LIN {X 0,Y 516.535,Z 181.809,A -85,B 0,C 180,E1 -4926.761,E2 -4926.761} C_VEL
LIN {X 0,Y 516.469,Z 186.856,A -85,B 0,C 180,E1 -4929.874,E2 -4929.874} C_VEL
LIN {X 0,Y 516.401,Z 191.39,A -85,B 0,C 180,E1 -4932.578,E2 -4932.578} C_VEL
LIN {X 0,Y 516.332,Z 197.348,A -85,B 0,C 180,E1 -4936.019,E2 -4936.019} C_VEL
LIN {X 0,Y 516.35,Z 197.756,A -85,B 0,C 180,E1 -4936.183,E2 -4936.183} C_VEL
LIN {X 0,Y 518.498,Z 209.145,A -85,B 0,C 180,E1 -4936.528,E2 -4936.528} C_VEL
LIN {X 0,Y 518.233,Z 222.389,A -85,B 0,C 180,E1 -4937.02,E2 -4937.02} C_VEL
LIN {X 0,Y 517.941,Z 233.553,A -85,B 0,C 180,E1 -4937.583,E2 -4937.583} C_VEL
LIN {X 0,Y 517.678,Z 245.305,A -85,B 0,C 180,E1 -4938.35,E2 -4938.35} C_VEL
LIN {X 0,Y 517.363,Z 255.999,A -85,B 0,C 180,E1 -4939.235,E2 -4939.235} C_VEL
LIN {X 0,Y 517.09,Z 265.619,A -85,B 0,C 180,E1 -4940.219,E2 -4940.219} C_VEL
LIN {X 0,Y 516.888,Z 273.497,A -85,B 0,C 180,E1 -4941.202,E2 -4941.202} C_VEL
LIN {X 0,Y 516.632,Z 281.203,A -85,B 0,C 180,E1 -4942.378,E2 -4942.378} C_VEL
LIN {X 0,Y 516.521,Z 288.266,A -85,B 0,C 180,E1 -4943.751,E2 -4943.751} C_VEL
LIN {X 0,Y 516.313,Z 292.978,A -85,B 0,C 180,E1 -4944.924,E2 -4944.924} C_VEL
LIN {X 0,Y 516.373,Z 296.581,A -85,B 0,C 180,E1 -4946.098,E2 -4946.098} C_VEL
LIN {X 0,Y 516.327,Z 298.446,A -85,B 0,C 180,E1 -4946.879,E2 -4946.879} C_VEL
LIN {X 0,Y 516.266,Z 299.854,A -85,B 0,C 180,E1 -4947.66,E2 -4947.66} C_VEL
LIN {X 0,Y 516.162,Z 301.473,A -85,B 0,C 180,E1 -4949.22,E2 -4949.22} C_VEL
LIN {X 0,Y 516.158,Z 301.71,A -85,B 0,C 180,E1 -4950,E2 -4950} C_VEL
LIN {X 0,Y 516.162,Z 301.527,A -85,B 0,C 180,E1 -4950.78,E2 -4950.78} C_VEL
LIN {X 0,Y 516.266,Z 299.979,A -85,B 0,C 180,E1 -4952.341,E2 -4952.341} C_VEL
LIN {X 0,Y 516.327,Z 298.625,A -85,B 0,C 180,E1 -4953.121,E2 -4953.121} C_VEL
LIN {X 0,Y 516.366,Z 295.765,A -85,B 0,C 180,E1 -4954.293,E2 -4954.293} C_VEL
LIN {X 0,Y 516.406,Z 291.887,A -85,B 0,C 180,E1 -4955.467,E2 -4955.467} C_VEL
LIN {X 0,Y 516.501,Z 285.975,A -85,B 0,C 180,E1 -4956.826,E2 -4956.826} C_VEL
LIN {X 0,Y 516.689,Z 279.36,A -85,B 0,C 180,E1 -4958.014,E2 -4958.014} C_VEL
LIN {X 0,Y 516.918,Z 271.215,A -85,B 0,C 180,E1 -4959.193,E2 -4959.193} C_VEL
LIN {X 0,Y 517.183,Z 262.876,A -85,B 0,C 180,E1 -4960.175,E2 -4960.175} C_VEL
LIN {X 0,Y 517.449,Z 252.583,A -85,B 0,C 180,E1 -4961.16,E2 -4961.16} C_VEL
LIN {X 0,Y 517.786,Z 240.919,A -85,B 0,C 180,E1 -4962.049,E2 -4962.049} C_VEL
LIN {X 0,Y 518.096,Z 229.411,A -85,B 0,C 180,E1 -4962.735,E2 -4962.735} C_VEL
LIN {X 0,Y 518.366,Z 217.395,A -85,B 0,C 180,E1 -4963.276,E2 -4963.276} C_VEL
LIN {X 0,Y 518.295,Z 207.984,A -85,B 0,C 180,E1 -4963.602,E2 -4963.602} C_VEL
LIN {X 0,Y 516.35,Z 197.574,A -85,B 0,C 180,E1 -4963.931,E2 -4963.931} C_VEL
LIN {X 0,Y 516.402,Z 191.56,A -85,B 0,C 180,E1 -4967.422,E2 -4967.422} C_VEL
LIN {X 0,Y 516.456,Z 186.035,A -85,B 0,C 180,E1 -4970.721,E2 -4970.721} C_VEL
LIN {X 0,Y 516.533,Z 181.956,A -85,B 0,C 180,E1 -4973.24,E2 -4973.24} C_VEL
LIN {X 0,Y 516.595,Z 177.386,A -85,B 0,C 180,E1 -4976.117,E2 -4976.117} C_VEL
LIN {X 0,Y 516.706,Z 172.392,A -85,B 0,C 180,E1 -4979.318,E2 -4979.318} C_VEL
LIN {X 0,Y 516.761,Z 167.51,A -85,B 0,C 180,E1 -4982.519,E2 -4982.519} C_VEL
LIN {X 0,Y 516.796,Z 163.328,A -85,B 0,C 180,E1 -4985.318,E2 -4985.318} C_VEL
LIN {X 0,Y 516.855,Z 163.102,A -85,B 0,C 180,E1 -4987.939,E2 -4987.939} C_VEL
LIN {X 0,Y 516.855,Z 163.105,A -85,B 0,C 180,E1 -4990.744,E2 -4990.744} C_VEL
LIN {X 0,Y 516.859,Z 163.102,A -85,B 0,C 180,E1 -4992.834,E2 -4992.834} C_VEL
LIN {X 0,Y 516.897,Z 163.098,A -85,B 0,C 180,E1 -4995.007,E2 -4995.007} C_VEL
LIN {X 0,Y 516.915,Z 163.094,A -85,B 0,C 180,E1 -4998.399,E2 -4998.399} C_VEL
LIN {X 0,Y 516.877,Z 163.099,A -85,B 0,C 180,E1 -5001.283,E2 -5001.283} C_VEL
LIN {X 0,Y 516.852,Z 163.103,A -85,B 0,C 180,E1 -5004.673,E2 -5004.673} C_VEL
LIN {X 0,Y 516.895,Z 163.1,A -85,B 0,C 180,E1 -5007.457,E2 -5007.457} C_VEL
LIN {X 0,Y 516.923,Z 163.097,A -85,B 0,C 180,E1 -5010.695,E2 -5010.695} C_VEL
LIN {X 0,Y 516.944,Z 163.09,A -85,B 0,C 180,E1 -5013.804,E2 -5013.804} C_VEL
LIN {X 0,Y 516.859,Z 163.101,A -85,B 0,C 180,E1 -5016.776,E2 -5016.776} C_VEL
LIN {X 0,Y 516.94,Z 163.095,A -85,B 0,C 180,E1 -5019.732,E2 -5019.732} C_VEL
LIN {X 0,Y 516.908,Z 163.098,A -85,B 0,C 180,E1 -5022.595,E2 -5022.595} C_VEL
LIN {X 0,Y 516.944,Z 163.093,A -85,B 0,C 180,E1 -5025.03,E2 -5025.03} C_VEL
LIN {X 0,Y 516.967,Z 163.09,A -85,B 0,C 180,E1 -5028.234,E2 -5028.234} C_VEL
LIN {X 0,Y 516.93,Z 163.096,A -85,B 0,C 180,E1 -5031.399,E2 -5031.399} C_VEL
LIN {X 0,Y 517.008,Z 163.084,A -85,B 0,C 180,E1 -5034.54,E2 -5034.54} C_VEL
LIN {X 0,Y 517.08,Z 163.074,A -85,B 0,C 180,E1 -5037.663,E2 -5037.663} C_VEL
LIN {X 0,Y 517.095,Z 163.072,A -85,B 0,C 180,E1 -5040.779,E2 -5040.779} C_VEL
LIN {X 0,Y 517.011,Z 163.085,A -85,B 0,C 180,E1 -5043.117,E2 -5043.117} C_VEL
LIN {X 0,Y 516.973,Z 163.086,A -85,B 0,C 180,E1 -5046.244,E2 -5046.244} C_VEL
LIN {X 0,Y 516.933,Z 163.091,A -85,B 0,C 180,E1 -5049.39,E2 -5049.39} C_VEL
LIN {X 0,Y 516.985,Z 163.088,A -85,B 0,C 180,E1 -5051.824,E2 -5051.824} C_VEL
LIN {X 0,Y 516.946,Z 163.094,A -85,B 0,C 180,E1 -5055.146,E2 -5055.146} C_VEL
LIN {X 0,Y 516.917,Z 163.095,A -85,B 0,C 180,E1 -5058.223,E2 -5058.223} C_VEL
LIN {X 0,Y 516.913,Z 163.098,A -85,B 0,C 180,E1 -5060.702,E2 -5060.702} C_VEL
LIN {X 0,Y 516.89,Z 163.103,A -85,B 0,C 180,E1 -5064.073,E2 -5064.073} C_VEL
LIN {X 0,Y 516.923,Z 163.093,A -85,B 0,C 180,E1 -5066.658,E2 -5066.658} C_VEL
LIN {X 0,Y 516.912,Z 163.098,A -85,B 0,C 180,E1 -5069.524,E2 -5069.524} C_VEL
LIN {X 0,Y 516.897,Z 163.1,A -85,B 0,C 180,E1 -5072.543,E2 -5072.543} C_VEL
LIN {X 0,Y 516.854,Z 163.102,A -85,B 0,C 180,E1 -5075.328,E2 -5075.328} C_VEL
LIN {X 0,Y 516.872,Z 163.098,A -85,B 0,C 180,E1 -5078.717,E2 -5078.717} C_VEL
LIN {X 0,Y 516.913,Z 163.095,A -85,B 0,C 180,E1 -5081.775,E2 -5081.775} C_VEL
LIN {X 0,Y 516.896,Z 163.099,A -85,B 0,C 180,E1 -5085.007,E2 -5085.007} C_VEL
LIN {X 0,Y 516.915,Z 163.097,A -85,B 0,C 180,E1 -5088.399,E2 -5088.399} C_VEL
LIN {X 0,Y 516.877,Z 163.105,A -85,B 0,C 180,E1 -5091.284,E2 -5091.284} C_VEL
LIN {X 0,Y 516.893,Z 163.21,A -85,B 0,C 180,E1 -5092.277,E2 -5092.277} C_VEL
LIN {X 0,Y 517.603,Z 168.389,A -85,B 0,C 180,E1 -5094.556,E2 -5094.556} C_VEL
LIN {X 0,Y 517.467,Z 175.12,A -85,B 0,C 180,E1 -5097.358,E2 -5097.358} C_VEL
LIN {X 0,Y 517.281,Z 182.741,A -85,B 0,C 180,E1 -5100.405,E2 -5100.405} C_VEL
LIN {X 0,Y 517.087,Z 190.334,A -85,B 0,C 180,E1 -5103.351,E2 -5103.351} C_VEL
LIN {X 0,Y 516.934,Z 198.126,A -85,B 0,C 180,E1 -5106.355,E2 -5106.355} C_VEL
LIN {X 0,Y 516.785,Z 205.917,A -85,B 0,C 180,E1 -5109.293,E2 -5109.293} C_VEL
LIN {X 0,Y 516.635,Z 213.829,A -85,B 0,C 180,E1 -5112.221,E2 -5112.221} C_VEL
LIN {X 0,Y 516.548,Z 221.5,A -85,B 0,C 180,E1 -5115.018,E2 -5115.018} C_VEL
LIN {X 0,Y 516.504,Z 224.491,A -85,B 0,C 180,E1 -5116.099,E2 -5116.099} C_VEL
LIN {X 0,Y 518.468,Z 237.09,A -85,B 0,C 180,E1 -5116.452,E2 -5116.452} C_VEL
LIN {X 0,Y 518.229,Z 250.11,A -85,B 0,C 180,E1 -5116.92,E2 -5116.92} C_VEL
LIN {X 0,Y 517.912,Z 262.468,A -85,B 0,C 180,E1 -5117.533,E2 -5117.533} C_VEL
LIN {X 0,Y 517.621,Z 273.585,A -85,B 0,C 180,E1 -5118.249,E2 -5118.249} C_VEL
LIN {X 0,Y 517.322,Z 284.469,A -85,B 0,C 180,E1 -5119.135,E2 -5119.135} C_VEL
LIN {X 0,Y 517.038,Z 293.333,A -85,B 0,C 180,E1 -5120.02,E2 -5120.02} C_VEL
LIN {X 0,Y 516.814,Z 302.959,A -85,B 0,C 180,E1 -5121.2,E2 -5121.2} C_VEL
LIN {X 0,Y 516.563,Z 310.62,A -85,B 0,C 180,E1 -5122.377,E2 -5122.377} C_VEL
LIN {X 0,Y 516.427,Z 317.679,A -85,B 0,C 180,E1 -5123.75,E2 -5123.75} C_VEL
LIN {X 0,Y 516.313,Z 322.372,A -85,B 0,C 180,E1 -5124.924,E2 -5124.924} C_VEL
LIN {X 0,Y 516.355,Z 325.957,A -85,B 0,C 180,E1 -5126.098,E2 -5126.098} C_VEL
LIN {X 0,Y 516.282,Z 327.807,A -85,B 0,C 180,E1 -5126.878,E2 -5126.878} C_VEL
LIN {X 0,Y 516.261,Z 329.196,A -85,B 0,C 180,E1 -5127.659,E2 -5127.659} C_VEL
LIN {X 0,Y 516.16,Z 330.785,A -85,B 0,C 180,E1 -5129.22,E2 -5129.22} C_VEL
LIN {X 0,Y 516.154,Z 331,A -85,B 0,C 180,E1 -5130,E2 -5130} C_VEL
LIN {X 0,Y 516.192,Z 330.186,A -85,B 0,C 180,E1 -5131.56,E2 -5131.56} C_VEL
LIN {X 0,Y 516.261,Z 329.198,A -85,B 0,C 180,E1 -5132.34,E2 -5132.34} C_VEL
LIN {X 0,Y 516.282,Z 327.81,A -85,B 0,C 180,E1 -5133.121,E2 -5133.121} C_VEL
LIN {X 0,Y 516.343,Z 324.896,A -85,B 0,C 180,E1 -5134.293,E2 -5134.293} C_VEL
LIN {X 0,Y 516.405,Z 320.949,A -85,B 0,C 180,E1 -5135.466,E2 -5135.466} C_VEL
LIN {X 0,Y 516.487,Z 315.031,A -85,B 0,C 180,E1 -5136.808,E2 -5136.808} C_VEL
LIN {X 0,Y 516.64,Z 308.238,A -85,B 0,C 180,E1 -5138.015,E2 -5138.015} C_VEL
LIN {X 0,Y 516.867,Z 299.993,A -85,B 0,C 180,E1 -5139.193,E2 -5139.193} C_VEL
LIN {X 0,Y 517.076,Z 291.541,A -85,B 0,C 180,E1 -5140.177,E2 -5140.177} C_VEL
LIN {X 0,Y 517.44,Z 281.099,A -85,B 0,C 180,E1 -5141.16,E2 -5141.16} C_VEL
LIN {X 0,Y 517.705,Z 269.737,A -85,B 0,C 180,E1 -5142.019,E2 -5142.019} C_VEL
LIN {X 0,Y 517.977,Z 259.412,A -85,B 0,C 180,E1 -5142.638,E2 -5142.638} C_VEL
LIN {X 0,Y 518.279,Z 247.77,A -85,B 0,C 180,E1 -5143.178,E2 -5143.178} C_VEL
LIN {X 0,Y 518.366,Z 235.727,A -85,B 0,C 180,E1 -5143.588,E2 -5143.588} C_VEL
LIN {X 0,Y 516.504,Z 224.492,A -85,B 0,C 180,E1 -5143.901,E2 -5143.901} C_VEL
LIN {X 0,Y 516.615,Z 215.936,A -85,B 0,C 180,E1 -5147.006,E2 -5147.006} C_VEL
LIN {X 0,Y 516.791,Z 207.212,A -85,B 0,C 180,E1 -5150.223,E2 -5150.223} C_VEL
LIN {X 0,Y 516.909,Z 199.24,A -85,B 0,C 180,E1 -5153.221,E2 -5153.221} C_VEL
LIN {X 0,Y 517.077,Z 191.419,A -85,B 0,C 180,E1 -5156.226,E2 -5156.226} C_VEL
LIN {X 0,Y 517.262,Z 183.54,A -85,B 0,C 180,E1 -5159.283,E2 -5159.283} C_VEL
LIN {X 0,Y 517.402,Z 176.722,A -85,B 0,C 180,E1 -5161.988,E2 -5161.988} C_VEL
LIN {X 0,Y 517.61,Z 169.972,A -85,B 0,C 180,E1 -5164.768,E2 -5164.768} C_VEL
LIN {X 0,Y 517.286,Z 165.445,A -85,B 0,C 180,E1 -5166.717,E2 -5166.717} C_VEL
LIN {X 0,Y 516.878,Z 163.104,A -85,B 0,C 180,E1 -5167.8,E2 -5167.8} C_VEL
LIN {X 0,Y 516.882,Z 163.102,A -85,B 0,C 180,E1 -5170.741,E2 -5170.741} C_VEL
LIN {X 0,Y 516.883,Z 163.099,A -85,B 0,C 180,E1 -5172.831,E2 -5172.831} C_VEL
LIN {X 0,Y 516.894,Z 163.099,A -85,B 0,C 180,E1 -5175.007,E2 -5175.007} C_VEL
LIN {X 0,Y 516.912,Z 163.096,A -85,B 0,C 180,E1 -5178.398,E2 -5178.398} C_VEL
LIN {X 0,Y 516.873,Z 163.098,A -85,B 0,C 180,E1 -5181.283,E2 -5181.283} C_VEL
LIN {X 0,Y 516.853,Z 163.102,A -85,B 0,C 180,E1 -5184.672,E2 -5184.672} C_VEL
LIN {X 0,Y 516.894,Z 163.1,A -85,B 0,C 180,E1 -5187.456,E2 -5187.456} C_VEL
LIN {X 0,Y 516.921,Z 163.098,A -85,B 0,C 180,E1 -5190.695,E2 -5190.695} C_VEL
LIN {X 0,Y 516.941,Z 163.092,A -85,B 0,C 180,E1 -5193.804,E2 -5193.804} C_VEL
LIN {X 0,Y 516.856,Z 163.1,A -85,B 0,C 180,E1 -5196.776,E2 -5196.776} C_VEL
LIN {X 0,Y 516.937,Z 163.094,A -85,B 0,C 180,E1 -5199.732,E2 -5199.732} C_VEL
LIN {X 0,Y 516.919,Z 163.097,A -85,B 0,C 180,E1 -5202.596,E2 -5202.596} C_VEL
LIN {X 0,Y 516.94,Z 163.093,A -85,B 0,C 180,E1 -5205.03,E2 -5205.03} C_VEL
LIN {X 0,Y 516.964,Z 163.091,A -85,B 0,C 180,E1 -5208.234,E2 -5208.234} C_VEL
LIN {X 0,Y 516.926,Z 163.098,A -85,B 0,C 180,E1 -5211.399,E2 -5211.399} C_VEL
LIN {X 0,Y 517.01,Z 163.084,A -85,B 0,C 180,E1 -5214.54,E2 -5214.54} C_VEL
LIN {X 0,Y 517.08,Z 163.074,A -85,B 0,C 180,E1 -5217.663,E2 -5217.663} C_VEL
LIN {X 0,Y 517.092,Z 163.073,A -85,B 0,C 180,E1 -5220.779,E2 -5220.779} C_VEL
LIN {X 0,Y 517.008,Z 163.086,A -85,B 0,C 180,E1 -5223.117,E2 -5223.117} C_VEL
LIN {X 0,Y 516.969,Z 163.088,A -85,B 0,C 180,E1 -5226.244,E2 -5226.244} C_VEL
LIN {X 0,Y 516.934,Z 163.09,A -85,B 0,C 180,E1 -5229.39,E2 -5229.39} C_VEL
LIN {X 0,Y 516.95,Z 163.092,A -85,B 0,C 180,E1 -5231.807,E2 -5231.807} C_VEL
LIN {X 0,Y 516.943,Z 163.094,A -85,B 0,C 180,E1 -5235.147,E2 -5235.147} C_VEL
LIN {X 0,Y 516.923,Z 163.094,A -85,B 0,C 180,E1 -5238.222,E2 -5238.222} C_VEL
LIN {X 0,Y 516.91,Z 163.098,A -85,B 0,C 180,E1 -5240.702,E2 -5240.702} C_VEL
LIN {X 0,Y 516.888,Z 163.101,A -85,B 0,C 180,E1 -5244.073,E2 -5244.073} C_VEL
LIN {X 0,Y 516.924,Z 163.092,A -85,B 0,C 180,E1 -5246.658,E2 -5246.658} C_VEL
LIN {X 0,Y 516.91,Z 163.097,A -85,B 0,C 180,E1 -5249.524,E2 -5249.524} C_VEL
LIN {X 0,Y 516.894,Z 163.1,A -85,B 0,C 180,E1 -5252.544,E2 -5252.544} C_VEL
LIN {X 0,Y 516.853,Z 163.103,A -85,B 0,C 180,E1 -5255.328,E2 -5255.328} C_VEL
LIN {X 0,Y 516.874,Z 163.099,A -85,B 0,C 180,E1 -5258.717,E2 -5258.717} C_VEL
LIN {X 0,Y 516.911,Z 163.094,A -85,B 0,C 180,E1 -5261.776,E2 -5261.776} C_VEL
LIN {X 0,Y 516.923,Z 163.095,A -85,B 0,C 180,E1 -5265.01,E2 -5265.01} C_VEL
LIN {X 0,Y 516.913,Z 163.097,A -85,B 0,C 180,E1 -5268.399,E2 -5268.399} C_VEL
LIN {X 0,Y 516.861,Z 163.102,A -85,B 0,C 180,E1 -5270.288,E2 -5270.288} C_VEL
LIN {X 0,Y 516.201,Z 163.187,A -85,B 0,C 180,E1 -5270.939,E2 -5270.939} C_VEL
LIN {X 0,Y 513.362,Z 163.539,A -85,B 0,C 180,E1 -5271.994,E2 -5271.994} C_VEL
LIN {X 0,Y 510.94,Z 163.842,A -85,B 0,C 180,E1 -5272.845,E2 -5272.845} C_VEL
LIN {X 0,Y 509.871,Z 163.975,A -85,B 0,C 180,E1 -5273.501,E2 -5273.501} C_VEL
LIN {X 0,Y 509.769,Z 163.986,A -85,B 0,C 180,E1 -5273.724,E2 -5273.724} C_VEL
LIN {X 0,Y 509.728,Z 163.995,A -85,B 0,C 180,E1 -5274.614,E2 -5274.614} C_VEL
LIN {X 0,Y 509.723,Z 168.189,A -85,B 0,C 180,E1 -5277.471,E2 -5277.471} C_VEL
LIN {X 0,Y 509.636,Z 172.476,A -85,B 0,C 180,E1 -5280.318,E2 -5280.318} C_VEL
LIN {X 0,Y 509.553,Z 176.479,A -85,B 0,C 180,E1 -5282.926,E2 -5282.926} C_VEL
LIN {X 0,Y 509.555,Z 180.576,A -85,B 0,C 180,E1 -5285.558,E2 -5285.558} C_VEL
LIN {X 0,Y 509.424,Z 184.667,A -85,B 0,C 180,E1 -5288.131,E2 -5288.131} C_VEL
LIN {X 0,Y 509.328,Z 188.766,A -85,B 0,C 180,E1 -5290.661,E2 -5290.661} C_VEL
LIN {X 0,Y 509.278,Z 192.925,A -85,B 0,C 180,E1 -5293.154,E2 -5293.154} C_VEL
LIN {X 0,Y 509.251,Z 197.77,A -85,B 0,C 180,E1 -5295.974,E2 -5295.974} C_VEL
LIN {X 0,Y 511.595,Z 210.137,A -85,B 0,C 180,E1 -5296.368,E2 -5296.368} C_VEL
LIN {X 0,Y 511.296,Z 223.744,A -85,B 0,C 180,E1 -5296.892,E2 -5296.892} C_VEL
LIN {X 0,Y 511.018,Z 235.001,A -85,B 0,C 180,E1 -5297.482,E2 -5297.482} C_VEL
LIN {X 0,Y 510.737,Z 245.526,A -85,B 0,C 180,E1 -5298.189,E2 -5298.189} C_VEL
LIN {X 0,Y 510.398,Z 256.219,A -85,B 0,C 180,E1 -5299.086,E2 -5299.086} C_VEL
LIN {X 0,Y 510.098,Z 265.838,A -85,B 0,C 180,E1 -5300.083,E2 -5300.083} C_VEL
LIN {X 0,Y 509.88,Z 273.715,A -85,B 0,C 180,E1 -5301.08,E2 -5301.08} C_VEL
LIN {X 0,Y 509.603,Z 281.42,A -85,B 0,C 180,E1 -5302.273,E2 -5302.273} C_VEL
LIN {X 0,Y 509.443,Z 288.483,A -85,B 0,C 180,E1 -5303.664,E2 -5303.664} C_VEL
LIN {X 0,Y 509.248,Z 293.194,A -85,B 0,C 180,E1 -5304.854,E2 -5304.854} C_VEL
LIN {X 0,Y 509.305,Z 296.796,A -85,B 0,C 180,E1 -5306.044,E2 -5306.044} C_VEL
LIN {X 0,Y 509.241,Z 298.66,A -85,B 0,C 180,E1 -5306.836,E2 -5306.836} C_VEL
LIN {X 0,Y 509.196,Z 300.067,A -85,B 0,C 180,E1 -5307.627,E2 -5307.627} C_VEL
LIN {X 0,Y 509.076,Z 301.686,A -85,B 0,C 180,E1 -5309.209,E2 -5309.209} C_VEL
LIN {X 0,Y 509.069,Z 301.923,A -85,B 0,C 180,E1 -5310,E2 -5310} C_VEL
LIN {X 0,Y 509.075,Z 301.739,A -85,B 0,C 180,E1 -5310.791,E2 -5310.791} C_VEL
LIN {X 0,Y 509.196,Z 300.191,A -85,B 0,C 180,E1 -5312.373,E2 -5312.373} C_VEL
LIN {X 0,Y 509.242,Z 298.837,A -85,B 0,C 180,E1 -5313.165,E2 -5313.165} C_VEL
LIN {X 0,Y 509.289,Z 295.977,A -85,B 0,C 180,E1 -5314.353,E2 -5314.353} C_VEL
LIN {X 0,Y 509.351,Z 292.097,A -85,B 0,C 180,E1 -5315.543,E2 -5315.543} C_VEL
LIN {X 0,Y 509.431,Z 286.405,A -85,B 0,C 180,E1 -5316.878,E2 -5316.878} C_VEL
LIN {X 0,Y 509.655,Z 279.569,A -85,B 0,C 180,E1 -5318.126,E2 -5318.126} C_VEL
LIN {X 0,Y 509.911,Z 271.423,A -85,B 0,C 180,E1 -5319.32,E2 -5319.32} C_VEL
LIN {X 0,Y 510.181,Z 263.084,A -85,B 0,C 180,E1 -5320.316,E2 -5320.316} C_VEL
LIN {X 0,Y 510.491,Z 252.788,A -85,B 0,C 180,E1 -5321.314,E2 -5321.314} C_VEL
LIN {X 0,Y 510.819,Z 241.691,A -85,B 0,C 180,E1 -5322.175,E2 -5322.175} C_VEL
LIN {X 0,Y 511.135,Z 231.426,A -85,B 0,C 180,E1 -5322.81,E2 -5322.81} C_VEL
LIN {X 0,Y 511.41,Z 220.114,A -85,B 0,C 180,E1 -5323.359,E2 -5323.359} C_VEL
LIN {X 0,Y 511.429,Z 209.032,A -85,B 0,C 180,E1 -5323.763,E2 -5323.763} C_VEL
LIN {X 0,Y 509.273,Z 197.748,A -85,B 0,C 180,E1 -5324.128,E2 -5324.128} C_VEL
LIN {X 0,Y 509.352,Z 191.695,A -85,B 0,C 180,E1 -5327.671,E2 -5327.671} C_VEL
LIN {X 0,Y 509.399,Z 186.178,A -85,B 0,C 180,E1 -5331.021,E2 -5331.021} C_VEL
LIN {X 0,Y 509.471,Z 182.096,A -85,B 0,C 180,E1 -5333.581,E2 -5333.581} C_VEL
LIN {X 0,Y 509.53,Z 177.843,A -85,B 0,C 180,E1 -5336.291,E2 -5336.291} C_VEL
LIN {X 0,Y 509.61,Z 173.872,A -85,B 0,C 180,E1 -5338.861,E2 -5338.861} C_VEL
LIN {X 0,Y 509.661,Z 169.728,A -85,B 0,C 180,E1 -5341.601,E2 -5341.601} C_VEL
LIN {X 0,Y 509.759,Z 165.526,A -85,B 0,C 180,E1 -5344.421,E2 -5344.421} C_VEL
LIN {X 0,Y 509.761,Z 163.99,A -85,B 0,C 180,E1 -5345.568,E2 -5345.568} C_VEL
LIN {X 0,Y 509.811,Z 163.982,A -85,B 0,C 180,E1 -5348.342,E2 -5348.342} C_VEL
LIN {X 0,Y 509.837,Z 163.977,A -85,B 0,C 180,E1 -5351.427,E2 -5351.427} C_VEL
LIN {X 0,Y 509.841,Z 163.976,A -85,B 0,C 180,E1 -5354.67,E2 -5354.67} C_VEL
LIN {X 0,Y 509.857,Z 163.972,A -85,B 0,C 180,E1 -5358.103,E2 -5358.103} C_VEL
LIN {X 0,Y 509.846,Z 163.979,A -85,B 0,C 180,E1 -5360.647,E2 -5360.647} C_VEL
LIN {X 0,Y 509.78,Z 163.985,A -85,B 0,C 180,E1 -5363.643,E2 -5363.643} C_VEL
LIN {X 0,Y 509.84,Z 163.977,A -85,B 0,C 180,E1 -5366.537,E2 -5366.537} C_VEL
LIN {X 0,Y 509.847,Z 163.978,A -85,B 0,C 180,E1 -5369.334,E2 -5369.334} C_VEL
LIN {X 0,Y 509.894,Z 163.969,A -85,B 0,C 180,E1 -5372.054,E2 -5372.054} C_VEL
LIN {X 0,Y 509.841,Z 163.976,A -85,B 0,C 180,E1 -5374.702,E2 -5374.702} C_VEL
LIN {X 0,Y 509.826,Z 163.978,A -85,B 0,C 180,E1 -5377.458,E2 -5377.458} C_VEL
LIN {X 0,Y 509.918,Z 163.969,A -85,B 0,C 180,E1 -5379.845,E2 -5379.845} C_VEL
LIN {X 0,Y 509.876,Z 163.975,A -85,B 0,C 180,E1 -5383.174,E2 -5383.174} C_VEL
LIN {X 0,Y 509.865,Z 163.973,A -85,B 0,C 180,E1 -5385.634,E2 -5385.634} C_VEL
LIN {X 0,Y 509.912,Z 163.966,A -85,B 0,C 180,E1 -5388.874,E2 -5388.874} C_VEL
LIN {X 0,Y 509.876,Z 163.971,A -85,B 0,C 180,E1 -5392.077,E2 -5392.077} C_VEL
LIN {X 0,Y 509.959,Z 163.962,A -85,B 0,C 180,E1 -5394.464,E2 -5394.464} C_VEL
LIN {X 0,Y 510.052,Z 163.95,A -85,B 0,C 180,E1 -5397.631,E2 -5397.631} C_VEL
LIN {X 0,Y 510.065,Z 163.948,A -85,B 0,C 180,E1 -5400.789,E2 -5400.789} C_VEL
LIN {X 0,Y 509.952,Z 163.965,A -85,B 0,C 180,E1 -5403.16,E2 -5403.16} C_VEL
LIN {X 0,Y 509.921,Z 163.965,A -85,B 0,C 180,E1 -5406.33,E2 -5406.33} C_VEL
LIN {X 0,Y 509.874,Z 163.971,A -85,B 0,C 180,E1 -5409.521,E2 -5409.521} C_VEL
LIN {X 0,Y 509.953,Z 163.964,A -85,B 0,C 180,E1 -5411.931,E2 -5411.931} C_VEL
LIN {X 0,Y 509.895,Z 163.973,A -85,B 0,C 180,E1 -5415.242,E2 -5415.242} C_VEL
LIN {X 0,Y 509.868,Z 163.972,A -85,B 0,C 180,E1 -5417.993,E2 -5417.993} C_VEL
LIN {X 0,Y 509.887,Z 163.974,A -85,B 0,C 180,E1 -5420.401,E2 -5420.401} C_VEL
LIN {X 0,Y 509.822,Z 163.978,A -85,B 0,C 180,E1 -5423.564,E2 -5423.564} C_VEL
LIN {X 0,Y 509.91,Z 163.967,A -85,B 0,C 180,E1 -5426.378,E2 -5426.378} C_VEL
LIN {X 0,Y 509.877,Z 163.974,A -85,B 0,C 180,E1 -5428.844,E2 -5428.844} C_VEL
LIN {X 0,Y 509.821,Z 163.979,A -85,B 0,C 180,E1 -5431.59,E2 -5431.59} C_VEL
LIN {X 0,Y 509.846,Z 163.978,A -85,B 0,C 180,E1 -5434.414,E2 -5434.414} C_VEL
LIN {X 0,Y 509.78,Z 163.985,A -85,B 0,C 180,E1 -5437.344,E2 -5437.344} C_VEL
LIN {X 0,Y 509.838,Z 163.975,A -85,B 0,C 180,E1 -5440.382,E2 -5440.382} C_VEL
LIN {X 0,Y 509.824,Z 163.982,A -85,B 0,C 180,E1 -5443.062,E2 -5443.062} C_VEL
LIN {X 0,Y 509.824,Z 163.98,A -85,B 0,C 180,E1 -5445.793,E2 -5445.793} C_VEL
LIN {X 0,Y 509.857,Z 163.975,A -85,B 0,C 180,E1 -5448.575,E2 -5448.575} C_VEL
LIN {X 0,Y 509.853,Z 163.979,A -85,B 0,C 180,E1 -5451.975,E2 -5451.975} C_VEL
LIN {X 0,Y 510.431,Z 167.613,A -85,B 0,C 180,E1 -5453.697,E2 -5453.697} C_VEL
LIN {X 0,Y 510.577,Z 172.233,A -85,B 0,C 180,E1 -5455.679,E2 -5455.679} C_VEL
LIN {X 0,Y 510.368,Z 179.311,A -85,B 0,C 180,E1 -5458.624,E2 -5458.624} C_VEL
LIN {X 0,Y 510.186,Z 185.708,A -85,B 0,C 180,E1 -5461.175,E2 -5461.175} C_VEL
LIN {X 0,Y 510.005,Z 193.668,A -85,B 0,C 180,E1 -5464.273,E2 -5464.273} C_VEL
LIN {X 0,Y 509.847,Z 201.465,A -85,B 0,C 180,E1 -5467.296,E2 -5467.296} C_VEL
LIN {X 0,Y 509.712,Z 209.256,A -85,B 0,C 180,E1 -5470.256,E2 -5470.256} C_VEL
LIN {X 0,Y 509.507,Z 218.161,A -85,B 0,C 180,E1 -5473.574,E2 -5473.574} C_VEL
LIN {X 0,Y 509.443,Z 224.491,A -85,B 0,C 180,E1 -5475.902,E2 -5475.902} C_VEL
LIN {X 0,Y 511.562,Z 237.925,A -85,B 0,C 180,E1 -5476.291,E2 -5476.291} C_VEL
LIN {X 0,Y 511.291,Z 251.238,A -85,B 0,C 180,E1 -5476.79,E2 -5476.79} C_VEL
LIN {X 0,Y 510.959,Z 263.766,A -85,B 0,C 180,E1 -5477.436,E2 -5477.436} C_VEL
LIN {X 0,Y 510.62,Z 274.904,A -85,B 0,C 180,E1 -5478.186,E2 -5478.186} C_VEL
LIN {X 0,Y 510.295,Z 285.537,A -85,B 0,C 180,E1 -5479.084,E2 -5479.084} C_VEL
LIN {X 0,Y 510.002,Z 295.111,A -85,B 0,C 180,E1 -5480.081,E2 -5480.081} C_VEL
LIN {X 0,Y 509.76,Z 302.959,A -85,B 0,C 180,E1 -5481.077,E2 -5481.077} C_VEL
LIN {X 0,Y 509.522,Z 310.62,A -85,B 0,C 180,E1 -5482.271,E2 -5482.271} C_VEL
LIN {X 0,Y 509.336,Z 317.679,A -85,B 0,C 180,E1 -5483.662,E2 -5483.662} C_VEL
LIN {X 0,Y 509.248,Z 322.372,A -85,B 0,C 180,E1 -5484.853,E2 -5484.853} C_VEL
LIN {X 0,Y 509.253,Z 325.957,A -85,B 0,C 180,E1 -5486.043,E2 -5486.043} C_VEL
LIN {X 0,Y 509.2,Z 327.807,A -85,B 0,C 180,E1 -5486.835,E2 -5486.835} C_VEL
LIN {X 0,Y 509.161,Z 329.196,A -85,B 0,C 180,E1 -5487.627,E2 -5487.627} C_VEL
LIN {X 0,Y 509.073,Z 330.785,A -85,B 0,C 180,E1 -5489.209,E2 -5489.209} C_VEL
LIN {X 0,Y 509.065,Z 331,A -85,B 0,C 180,E1 -5490,E2 -5490} C_VEL
LIN {X 0,Y 509.112,Z 330.185,A -85,B 0,C 180,E1 -5491.582,E2 -5491.582} C_VEL
LIN {X 0,Y 509.161,Z 329.198,A -85,B 0,C 180,E1 -5492.373,E2 -5492.373} C_VEL
LIN {X 0,Y 509.2,Z 327.81,A -85,B 0,C 180,E1 -5493.165,E2 -5493.165} C_VEL
LIN {X 0,Y 509.234,Z 324.896,A -85,B 0,C 180,E1 -5494.353,E2 -5494.353} C_VEL
LIN {X 0,Y 509.345,Z 320.949,A -85,B 0,C 180,E1 -5495.542,E2 -5495.542} C_VEL
LIN {X 0,Y 509.41,Z 315.283,A -85,B 0,C 180,E1 -5496.853,E2 -5496.853} C_VEL
LIN {X 0,Y 509.585,Z 308.238,A -85,B 0,C 180,E1 -5498.127,E2 -5498.127} C_VEL
LIN {X 0,Y 509.846,Z 299.993,A -85,B 0,C 180,E1 -5499.321,E2 -5499.321} C_VEL
LIN {X 0,Y 510.065,Z 291.541,A -85,B 0,C 180,E1 -5500.318,E2 -5500.318} C_VEL
LIN {X 0,Y 510.468,Z 281.098,A -85,B 0,C 180,E1 -5501.314,E2 -5501.314} C_VEL
LIN {X 0,Y 510.737,Z 270.479,A -85,B 0,C 180,E1 -5502.133,E2 -5502.133} C_VEL
LIN {X 0,Y 511.049,Z 259.412,A -85,B 0,C 180,E1 -5502.812,E2 -5502.812} C_VEL
LIN {X 0,Y 511.371,Z 247.77,A -85,B 0,C 180,E1 -5503.359,E2 -5503.359} C_VEL
LIN {X 0,Y 511.408,Z 236.184,A -85,B 0,C 180,E1 -5503.763,E2 -5503.763} C_VEL
LIN {X 0,Y 509.442,Z 224.492,A -85,B 0,C 180,E1 -5504.097,E2 -5504.097} C_VEL
LIN {X 0,Y 509.541,Z 215.936,A -85,B 0,C 180,E1 -5507.25,E2 -5507.25} C_VEL
LIN {X 0,Y 509.731,Z 207.64,A -85,B 0,C 180,E1 -5510.353,E2 -5510.353} C_VEL
LIN {X 0,Y 509.888,Z 199.24,A -85,B 0,C 180,E1 -5513.56,E2 -5513.56} C_VEL
LIN {X 0,Y 510.037,Z 191.907,A -85,B 0,C 180,E1 -5516.406,E2 -5516.406} C_VEL
LIN {X 0,Y 510.24,Z 184.572,A -85,B 0,C 180,E1 -5519.273,E2 -5519.273} C_VEL
LIN {X 0,Y 510.392,Z 177.758,A -85,B 0,C 180,E1 -5522.014,E2 -5522.014} C_VEL
LIN {X 0,Y 510.618,Z 171.004,A -85,B 0,C 180,E1 -5524.833,E2 -5524.833} C_VEL
LIN {X 0,Y 510.454,Z 167.615,A -85,B 0,C 180,E1 -5526.301,E2 -5526.301} C_VEL
LIN {X 0,Y 509.851,Z 163.979,A -85,B 0,C 180,E1 -5528.024,E2 -5528.024} C_VEL
LIN {X 0,Y 509.855,Z 163.977,A -85,B 0,C 180,E1 -5531.425,E2 -5531.425} C_VEL
LIN {X 0,Y 509.838,Z 163.977,A -85,B 0,C 180,E1 -5534.67,E2 -5534.67} C_VEL
LIN {X 0,Y 509.854,Z 163.974,A -85,B 0,C 180,E1 -5538.103,E2 -5538.103} C_VEL
LIN {X 0,Y 509.842,Z 163.98,A -85,B 0,C 180,E1 -5540.647,E2 -5540.647} C_VEL
LIN {X 0,Y 509.778,Z 163.984,A -85,B 0,C 180,E1 -5543.643,E2 -5543.643} C_VEL
LIN {X 0,Y 509.856,Z 163.974,A -85,B 0,C 180,E1 -5546.539,E2 -5546.539} C_VEL
LIN {X 0,Y 509.844,Z 163.978,A -85,B 0,C 180,E1 -5549.334,E2 -5549.334} C_VEL
LIN {X 0,Y 509.892,Z 163.971,A -85,B 0,C 180,E1 -5552.054,E2 -5552.054} C_VEL
LIN {X 0,Y 509.838,Z 163.977,A -85,B 0,C 180,E1 -5554.702,E2 -5554.702} C_VEL
LIN {X 0,Y 509.823,Z 163.979,A -85,B 0,C 180,E1 -5557.458,E2 -5557.458} C_VEL
LIN {X 0,Y 509.914,Z 163.968,A -85,B 0,C 180,E1 -5559.845,E2 -5559.845} C_VEL
LIN {X 0,Y 509.88,Z 163.974,A -85,B 0,C 180,E1 -5563.175,E2 -5563.175} C_VEL
LIN {X 0,Y 509.862,Z 163.974,A -85,B 0,C 180,E1 -5565.634,E2 -5565.634} C_VEL
LIN {X 0,Y 509.909,Z 163.967,A -85,B 0,C 180,E1 -5568.874,E2 -5568.874} C_VEL
LIN {X 0,Y 509.873,Z 163.97,A -85,B 0,C 180,E1 -5572.077,E2 -5572.077} C_VEL
LIN {X 0,Y 509.96,Z 163.961,A -85,B 0,C 180,E1 -5574.464,E2 -5574.464} C_VEL
LIN {X 0,Y 510.051,Z 163.95,A -85,B 0,C 180,E1 -5577.631,E2 -5577.631} C_VEL
LIN {X 0,Y 510.062,Z 163.949,A -85,B 0,C 180,E1 -5580.79,E2 -5580.79} C_VEL
LIN {X 0,Y 509.95,Z 163.966,A -85,B 0,C 180,E1 -5583.16,E2 -5583.16} C_VEL
LIN {X 0,Y 509.917,Z 163.967,A -85,B 0,C 180,E1 -5586.33,E2 -5586.33} C_VEL
LIN {X 0,Y 509.875,Z 163.97,A -85,B 0,C 180,E1 -5589.521,E2 -5589.521} C_VEL
LIN {X 0,Y 509.902,Z 163.971,A -85,B 0,C 180,E1 -5591.932,E2 -5591.932} C_VEL
LIN {X 0,Y 509.892,Z 163.972,A -85,B 0,C 180,E1 -5595.242,E2 -5595.242} C_VEL
LIN {X 0,Y 509.88,Z 163.971,A -85,B 0,C 180,E1 -5597.999,E2 -5597.999} C_VEL
LIN {X 0,Y 509.848,Z 163.976,A -85,B 0,C 180,E1 -5601.002,E2 -5601.002} C_VEL
LIN {X 0,Y 509.819,Z 163.979,A -85,B 0,C 180,E1 -5603.564,E2 -5603.564} C_VEL
LIN {X 0,Y 509.91,Z 163.966,A -85,B 0,C 180,E1 -5606.379,E2 -5606.379} C_VEL
LIN {X 0,Y 509.875,Z 163.973,A -85,B 0,C 180,E1 -5608.845,E2 -5608.845} C_VEL
LIN {X 0,Y 509.819,Z 163.979,A -85,B 0,C 180,E1 -5611.59,E2 -5611.59} C_VEL
LIN {X 0,Y 509.843,Z 163.978,A -85,B 0,C 180,E1 -5614.414,E2 -5614.414} C_VEL
LIN {X 0,Y 509.781,Z 163.986,A -85,B 0,C 180,E1 -5617.344,E2 -5617.344} C_VEL
LIN {X 0,Y 509.837,Z 163.975,A -85,B 0,C 180,E1 -5620.383,E2 -5620.383} C_VEL
LIN {X 0,Y 509.822,Z 163.981,A -85,B 0,C 180,E1 -5623.062,E2 -5623.062} C_VEL
LIN {X 0,Y 509.83,Z 163.979,A -85,B 0,C 180,E1 -5625.793,E2 -5625.793} C_VEL
LIN {X 0,Y 509.855,Z 163.975,A -85,B 0,C 180,E1 -5628.575,E2 -5628.575} C_VEL
LIN {X 0,Y 509.847,Z 163.977,A -85,B 0,C 180,E1 -5631.787,E2 -5631.787} C_VEL
LIN {X 0,Y 509.769,Z 163.986,A -85,B 0,C 180,E1 -5633.724,E2 -5633.724} C_VEL
LIN {X 0,Y 509.056,Z 164.275,A -85,B 0,C 180,E1 -5634.382,E2 -5634.382} C_VEL
LIN {X 0,Y 506.184,Z 165.647,A -85,B 0,C 180,E1 -5635.441,E2 -5635.441} C_VEL
LIN {X 0,Y 503.773,Z 167.182,A -85,B 0,C 180,E1 -5636.291,E2 -5636.291} C_VEL
LIN {X 0,Y 502.732,Z 168.263,A -85,B 0,C 180,E1 -5636.948,E2 -5636.948} C_VEL
LIN {X 0,Y 502.642,Z 168.595,A -85,B 0,C 180,E1 -5637.171,E2 -5637.171} C_VEL
LIN {X 0,Y 502.588,Z 172.957,A -85,B 0,C 180,E1 -5640.111,E2 -5640.111} C_VEL
LIN {X 0,Y 502.519,Z 176.598,A -85,B 0,C 180,E1 -5642.515,E2 -5642.515} C_VEL
LIN {X 0,Y 502.49,Z 181.012,A -85,B 0,C 180,E1 -5645.384,E2 -5645.384} C_VEL
LIN {X 0,Y 502.389,Z 184.811,A -85,B 0,C 180,E1 -5647.809,E2 -5647.809} C_VEL
LIN {X 0,Y 502.29,Z 188.92,A -85,B 0,C 180,E1 -5650.379,E2 -5650.379} C_VEL
LIN {X 0,Y 502.223,Z 193.088,A -85,B 0,C 180,E1 -5652.911,E2 -5652.911} C_VEL
LIN {X 0,Y 502.195,Z 197.939,A -85,B 0,C 180,E1 -5655.772,E2 -5655.772} C_VEL
LIN {X 0,Y 504.719,Z 211.129,A -85,B 0,C 180,E1 -5656.205,E2 -5656.205} C_VEL
LIN {X 0,Y 504.384,Z 223.971,A -85,B 0,C 180,E1 -5656.709,E2 -5656.709} C_VEL
LIN {X 0,Y 504.084,Z 235.491,A -85,B 0,C 180,E1 -5657.324,E2 -5657.324} C_VEL
LIN {X 0,Y 503.759,Z 247.034,A -85,B 0,C 180,E1 -5658.125,E2 -5658.125} C_VEL
LIN {X 0,Y 503.395,Z 257.504,A -85,B 0,C 180,E1 -5659.035,E2 -5659.035} C_VEL
LIN {X 0,Y 503.111,Z 266.057,A -85,B 0,C 180,E1 -5659.944,E2 -5659.944} C_VEL
LIN {X 0,Y 502.868,Z 273.933,A -85,B 0,C 180,E1 -5660.954,E2 -5660.954} C_VEL
LIN {X 0,Y 502.549,Z 281.637,A -85,B 0,C 180,E1 -5662.163,E2 -5662.163} C_VEL
LIN {X 0,Y 502.361,Z 288.7,A -85,B 0,C 180,E1 -5663.574,E2 -5663.574} C_VEL
LIN {X 0,Y 502.187,Z 293.409,A -85,B 0,C 180,E1 -5664.781,E2 -5664.781} C_VEL
LIN {X 0,Y 502.238,Z 297.01,A -85,B 0,C 180,E1 -5665.988,E2 -5665.988} C_VEL
LIN {X 0,Y 502.16,Z 298.875,A -85,B 0,C 180,E1 -5666.791,E2 -5666.791} C_VEL
LIN {X 0,Y 502.128,Z 300.281,A -85,B 0,C 180,E1 -5667.594,E2 -5667.594} C_VEL
LIN {X 0,Y 501.992,Z 301.899,A -85,B 0,C 180,E1 -5669.198,E2 -5669.198} C_VEL
LIN {X 0,Y 501.984,Z 302.136,A -85,B 0,C 180,E1 -5670,E2 -5670} C_VEL
LIN {X 0,Y 501.992,Z 301.952,A -85,B 0,C 180,E1 -5670.802,E2 -5670.802} C_VEL
LIN {X 0,Y 502.128,Z 300.402,A -85,B 0,C 180,E1 -5672.407,E2 -5672.407} C_VEL
LIN {X 0,Y 502.16,Z 299.049,A -85,B 0,C 180,E1 -5673.209,E2 -5673.209} C_VEL
LIN {X 0,Y 502.214,Z 296.188,A -85,B 0,C 180,E1 -5674.414,E2 -5674.414} C_VEL
LIN {X 0,Y 502.299,Z 292.308,A -85,B 0,C 180,E1 -5675.621,E2 -5675.621} C_VEL
LIN {X 0,Y 502.356,Z 287.305,A -85,B 0,C 180,E1 -5676.829,E2 -5676.829} C_VEL
LIN {X 0,Y 502.58,Z 281.001,A -85,B 0,C 180,E1 -5678.039,E2 -5678.039} C_VEL
LIN {X 0,Y 502.827,Z 273.111,A -85,B 0,C 180,E1 -5679.25,E2 -5679.25} C_VEL
LIN {X 0,Y 503.163,Z 265.064,A -85,B 0,C 180,E1 -5680.259,E2 -5680.259} C_VEL
LIN {X 0,Y 503.468,Z 255.247,A -85,B 0,C 180,E1 -5681.27,E2 -5681.27} C_VEL
LIN {X 0,Y 503.8,Z 245.588,A -85,B 0,C 180,E1 -5682.079,E2 -5682.079} C_VEL
LIN {X 0,Y 504.08,Z 234.662,A -85,B 0,C 180,E1 -5682.816,E2 -5682.816} C_VEL
LIN {X 0,Y 504.457,Z 222.566,A -85,B 0,C 180,E1 -5683.444,E2 -5683.444} C_VEL
LIN {X 0,Y 504.608,Z 210.373,A -85,B 0,C 180,E1 -5683.914,E2 -5683.914} C_VEL
LIN {X 0,Y 502.202,Z 197.915,A -85,B 0,C 180,E1 -5684.331,E2 -5684.331} C_VEL
LIN {X 0,Y 502.255,Z 191.858,A -85,B 0,C 180,E1 -5687.929,E2 -5687.929} C_VEL
LIN {X 0,Y 502.325,Z 187.686,A -85,B 0,C 180,E1 -5690.474,E2 -5690.474} C_VEL
LIN {X 0,Y 502.393,Z 183.603,A -85,B 0,C 180,E1 -5693.06,E2 -5693.06} C_VEL
LIN {X 0,Y 502.445,Z 179.501,A -85,B 0,C 180,E1 -5695.697,E2 -5695.697} C_VEL
LIN {X 0,Y 502.558,Z 175.366,A -85,B 0,C 180,E1 -5698.39,E2 -5698.39} C_VEL
LIN {X 0,Y 502.606,Z 170.755,A -85,B 0,C 180,E1 -5701.463,E2 -5701.463} C_VEL
LIN {X 0,Y 502.714,Z 166.394,A -85,B 0,C 180,E1 -5704.429,E2 -5704.429} C_VEL
LIN {X 0,Y 502.736,Z 164.863,A -85,B 0,C 180,E1 -5705.824,E2 -5705.824} C_VEL
LIN {X 0,Y 502.778,Z 164.859,A -85,B 0,C 180,E1 -5708.978,E2 -5708.978} C_VEL
LIN {X 0,Y 502.776,Z 164.858,A -85,B 0,C 180,E1 -5712.195,E2 -5712.195} C_VEL
LIN {X 0,Y 502.788,Z 164.859,A -85,B 0,C 180,E1 -5715.47,E2 -5715.47} C_VEL
LIN {X 0,Y 502.821,Z 164.855,A -85,B 0,C 180,E1 -5718.934,E2 -5718.934} C_VEL
LIN {X 0,Y 502.762,Z 164.858,A -85,B 0,C 180,E1 -5722.043,E2 -5722.043} C_VEL
LIN {X 0,Y 502.787,Z 164.855,A -85,B 0,C 180,E1 -5725.033,E2 -5725.033} C_VEL
LIN {X 0,Y 502.784,Z 164.858,A -85,B 0,C 180,E1 -5727.915,E2 -5727.915} C_VEL
LIN {X 0,Y 502.826,Z 164.853,A -85,B 0,C 180,E1 -5730.712,E2 -5730.712} C_VEL
LIN {X 0,Y 502.864,Z 164.844,A -85,B 0,C 180,E1 -5733.439,E2 -5733.439} C_VEL
LIN {X 0,Y 502.776,Z 164.86,A -85,B 0,C 180,E1 -5736.085,E2 -5736.085} C_VEL
LIN {X 0,Y 502.784,Z 164.855,A -85,B 0,C 180,E1 -5738.689,E2 -5738.689} C_VEL
LIN {X 0,Y 502.827,Z 164.852,A -85,B 0,C 180,E1 -5741.248,E2 -5741.248} C_VEL
LIN {X 0,Y 502.85,Z 164.849,A -85,B 0,C 180,E1 -5744.6,E2 -5744.6} C_VEL
LIN {X 0,Y 502.878,Z 164.847,A -85,B 0,C 180,E1 -5748.039,E2 -5748.039} C_VEL
LIN {X 0,Y 502.85,Z 164.847,A -85,B 0,C 180,E1 -5751.156,E2 -5751.156} C_VEL
LIN {X 0,Y 502.912,Z 164.839,A -85,B 0,C 180,E1 -5754.386,E2 -5754.386} C_VEL
LIN {X 0,Y 503.022,Z 164.826,A -85,B 0,C 180,E1 -5757.598,E2 -5757.598} C_VEL
LIN {X 0,Y 503.029,Z 164.827,A -85,B 0,C 180,E1 -5760,E2 -5760} C_VEL
LIN {X 0,Y 503.024,Z 164.825,A -85,B 0,C 180,E1 -5762.402,E2 -5762.402} C_VEL
LIN {X 0,Y 502.916,Z 164.838,A -85,B 0,C 180,E1 -5765.614,E2 -5765.614} C_VEL
LIN {X 0,Y 502.847,Z 164.85,A -85,B 0,C 180,E1 -5768.844,E2 -5768.844} C_VEL
LIN {X 0,Y 502.895,Z 164.844,A -85,B 0,C 180,E1 -5772.1,E2 -5772.1} C_VEL
LIN {X 0,Y 502.85,Z 164.849,A -85,B 0,C 180,E1 -5775.4,E2 -5775.4} C_VEL
LIN {X 0,Y 502.827,Z 164.854,A -85,B 0,C 180,E1 -5778.752,E2 -5778.752} C_VEL
LIN {X 0,Y 502.784,Z 164.854,A -85,B 0,C 180,E1 -5781.311,E2 -5781.311} C_VEL
LIN {X 0,Y 502.775,Z 164.859,A -85,B 0,C 180,E1 -5783.915,E2 -5783.915} C_VEL
LIN {X 0,Y 502.865,Z 164.844,A -85,B 0,C 180,E1 -5786.566,E2 -5786.566} C_VEL
LIN {X 0,Y 502.825,Z 164.853,A -85,B 0,C 180,E1 -5789.288,E2 -5789.288} C_VEL
LIN {X 0,Y 502.784,Z 164.857,A -85,B 0,C 180,E1 -5792.085,E2 -5792.085} C_VEL
LIN {X 0,Y 502.791,Z 164.854,A -85,B 0,C 180,E1 -5794.967,E2 -5794.967} C_VEL
LIN {X 0,Y 502.763,Z 164.856,A -85,B 0,C 180,E1 -5798.481,E2 -5798.481} C_VEL
LIN {X 0,Y 502.821,Z 164.853,A -85,B 0,C 180,E1 -5801.066,E2 -5801.066} C_VEL
LIN {X 0,Y 502.787,Z 164.859,A -85,B 0,C 180,E1 -5804.53,E2 -5804.53} C_VEL
LIN {X 0,Y 502.796,Z 164.855,A -85,B 0,C 180,E1 -5807.861,E2 -5807.861} C_VEL
LIN {X 0,Y 502.78,Z 164.859,A -85,B 0,C 180,E1 -5810.247,E2 -5810.247} C_VEL
LIN {X 0,Y 502.841,Z 164.998,A -85,B 0,C 180,E1 -5811.918,E2 -5811.918} C_VEL
LIN {X 0,Y 503.524,Z 169.766,A -85,B 0,C 180,E1 -5814.111,E2 -5814.111} C_VEL
LIN {X 0,Y 503.547,Z 174.308,A -85,B 0,C 180,E1 -5816.063,E2 -5816.063} C_VEL
LIN {X 0,Y 503.311,Z 181.041,A -85,B 0,C 180,E1 -5818.892,E2 -5818.892} C_VEL
LIN {X 0,Y 503.147,Z 187.878,A -85,B 0,C 180,E1 -5821.646,E2 -5821.646} C_VEL
LIN {X 0,Y 502.967,Z 195.814,A -85,B 0,C 180,E1 -5824.775,E2 -5824.775} C_VEL
LIN {X 0,Y 502.768,Z 203.691,A -85,B 0,C 180,E1 -5827.826,E2 -5827.826} C_VEL
LIN {X 0,Y 502.593,Z 211.482,A -85,B 0,C 180,E1 -5830.815,E2 -5830.815} C_VEL
LIN {X 0,Y 502.441,Z 219.274,A -85,B 0,C 180,E1 -5833.754,E2 -5833.754} C_VEL
LIN {X 0,Y 502.367,Z 224.491,A -85,B 0,C 180,E1 -5835.699,E2 -5835.699} C_VEL
LIN {X 0,Y 504.625,Z 237.925,A -85,B 0,C 180,E1 -5836.099,E2 -5836.099} C_VEL
LIN {X 0,Y 504.398,Z 251.238,A -85,B 0,C 180,E1 -5836.606,E2 -5836.606} C_VEL
LIN {X 0,Y 504.029,Z 262.609,A -85,B 0,C 180,E1 -5837.192,E2 -5837.192} C_VEL
LIN {X 0,Y 503.711,Z 273.586,A -85,B 0,C 180,E1 -5837.919,E2 -5837.919} C_VEL
LIN {X 0,Y 503.371,Z 284.467,A -85,B 0,C 180,E1 -5838.83,E2 -5838.83} C_VEL
LIN {X 0,Y 503.023,Z 293.332,A -85,B 0,C 180,E1 -5839.739,E2 -5839.739} C_VEL
LIN {X 0,Y 502.704,Z 302.959,A -85,B 0,C 180,E1 -5840.951,E2 -5840.951} C_VEL
LIN {X 0,Y 502.47,Z 310.621,A -85,B 0,C 180,E1 -5842.162,E2 -5842.162} C_VEL
LIN {X 0,Y 502.275,Z 317.679,A -85,B 0,C 180,E1 -5843.573,E2 -5843.573} C_VEL
LIN {X 0,Y 502.186,Z 322.372,A -85,B 0,C 180,E1 -5844.781,E2 -5844.781} C_VEL
LIN {X 0,Y 502.152,Z 325.958,A -85,B 0,C 180,E1 -5845.987,E2 -5845.987} C_VEL
LIN {X 0,Y 502.121,Z 327.807,A -85,B 0,C 180,E1 -5846.79,E2 -5846.79} C_VEL
LIN {X 0,Y 502.066,Z 329.195,A -85,B 0,C 180,E1 -5847.593,E2 -5847.593} C_VEL
LIN {X 0,Y 501.99,Z 330.786,A -85,B 0,C 180,E1 -5849.198,E2 -5849.198} C_VEL
LIN {X 0,Y 501.98,Z 331,A -85,B 0,C 180,E1 -5850,E2 -5850} C_VEL
LIN {X 0,Y 502.036,Z 330.185,A -85,B 0,C 180,E1 -5851.604,E2 -5851.604} C_VEL
LIN {X 0,Y 502.066,Z 329.198,A -85,B 0,C 180,E1 -5852.407,E2 -5852.407} C_VEL
LIN {X 0,Y 502.121,Z 327.81,A -85,B 0,C 180,E1 -5853.209,E2 -5853.209} C_VEL
LIN {X 0,Y 502.128,Z 324.896,A -85,B 0,C 180,E1 -5854.415,E2 -5854.415} C_VEL
LIN {X 0,Y 502.26,Z 320.949,A -85,B 0,C 180,E1 -5855.621,E2 -5855.621} C_VEL
LIN {X 0,Y 502.335,Z 314.978,A -85,B 0,C 180,E1 -5857.011,E2 -5857.011} C_VEL
LIN {X 0,Y 502.542,Z 308.238,A -85,B 0,C 180,E1 -5858.241,E2 -5858.241} C_VEL
LIN {X 0,Y 502.811,Z 299.993,A -85,B 0,C 180,E1 -5859.453,E2 -5859.453} C_VEL
LIN {X 0,Y 503.058,Z 291.541,A -85,B 0,C 180,E1 -5860.464,E2 -5860.464} C_VEL
LIN {X 0,Y 503.495,Z 281.097,A -85,B 0,C 180,E1 -5861.473,E2 -5861.473} C_VEL
LIN {X 0,Y 503.794,Z 269.422,A -85,B 0,C 180,E1 -5862.378,E2 -5862.378} C_VEL
LIN {X 0,Y 504.159,Z 257.494,A -85,B 0,C 180,E1 -5863.092,E2 -5863.092} C_VEL
LIN {X 0,Y 504.545,Z 245.173,A -85,B 0,C 180,E1 -5863.646,E2 -5863.646} C_VEL
LIN {X 0,Y 504.416,Z 236.64,A -85,B 0,C 180,E1 -5863.945,E2 -5863.945} C_VEL
LIN {X 0,Y 502.366,Z 224.492,A -85,B 0,C 180,E1 -5864.3,E2 -5864.3} C_VEL
LIN {X 0,Y 502.467,Z 217.049,A -85,B 0,C 180,E1 -5867.081,E2 -5867.081} C_VEL
LIN {X 0,Y 502.661,Z 209.257,A -85,B 0,C 180,E1 -5870.032,E2 -5870.032} C_VEL
LIN {X 0,Y 502.837,Z 201.466,A -85,B 0,C 180,E1 -5873.038,E2 -5873.038} C_VEL
LIN {X 0,Y 502.975,Z 193.541,A -85,B 0,C 180,E1 -5876.113,E2 -5876.113} C_VEL
LIN {X 0,Y 503.157,Z 186.742,A -85,B 0,C 180,E1 -5878.808,E2 -5878.808} C_VEL
LIN {X 0,Y 503.406,Z 179.817,A -85,B 0,C 180,E1 -5881.612,E2 -5881.612} C_VEL
LIN {X 0,Y 503.628,Z 172.034,A -85,B 0,C 180,E1 -5884.9,E2 -5884.9} C_VEL
LIN {X 0,Y 503.271,Z 167.521,A -85,B 0,C 180,E1 -5886.904,E2 -5886.904} C_VEL
LIN {X 0,Y 502.816,Z 164.856,A -85,B 0,C 180,E1 -5888.217,E2 -5888.217} C_VEL
LIN {X 0,Y 502.819,Z 164.853,A -85,B 0,C 180,E1 -5891.066,E2 -5891.066} C_VEL
LIN {X 0,Y 502.785,Z 164.855,A -85,B 0,C 180,E1 -5894.53,E2 -5894.53} C_VEL
LIN {X 0,Y 502.794,Z 164.853,A -85,B 0,C 180,E1 -5897.86,E2 -5897.86} C_VEL
LIN {X 0,Y 502.786,Z 164.856,A -85,B 0,C 180,E1 -5900.245,E2 -5900.245} C_VEL
LIN {X 0,Y 502.718,Z 164.862,A -85,B 0,C 180,E1 -5903.048,E2 -5903.048} C_VEL
LIN {X 0,Y 502.801,Z 164.856,A -85,B 0,C 180,E1 -5906.006,E2 -5906.006} C_VEL
LIN {X 0,Y 502.794,Z 164.857,A -85,B 0,C 180,E1 -5908.857,E2 -5908.857} C_VEL
LIN {X 0,Y 502.843,Z 164.848,A -85,B 0,C 180,E1 -5911.705,E2 -5911.705} C_VEL
LIN {X 0,Y 502.82,Z 164.854,A -85,B 0,C 180,E1 -5914.323,E2 -5914.323} C_VEL
LIN {X 0,Y 502.8,Z 164.853,A -85,B 0,C 180,E1 -5917.298,E2 -5917.298} C_VEL
LIN {X 0,Y 502.822,Z 164.85,A -85,B 0,C 180,E1 -5920.4,E2 -5920.4} C_VEL
LIN {X 0,Y 502.828,Z 164.852,A -85,B 0,C 180,E1 -5922.931,E2 -5922.931} C_VEL
LIN {X 0,Y 502.843,Z 164.848,A -85,B 0,C 180,E1 -5925.429,E2 -5925.429} C_VEL
LIN {X 0,Y 502.873,Z 164.844,A -85,B 0,C 180,E1 -5928.717,E2 -5928.717} C_VEL
LIN {X 0,Y 502.845,Z 164.846,A -85,B 0,C 180,E1 -5931.966,E2 -5931.966} C_VEL
LIN {X 0,Y 502.913,Z 164.838,A -85,B 0,C 180,E1 -5934.386,E2 -5934.386} C_VEL
LIN {X 0,Y 503.021,Z 164.826,A -85,B 0,C 180,E1 -5937.598,E2 -5937.598} C_VEL
LIN {X 0,Y 503.026,Z 164.827,A -85,B 0,C 180,E1 -5940,E2 -5940} C_VEL
LIN {X 0,Y 503.02,Z 164.826,A -85,B 0,C 180,E1 -5942.402,E2 -5942.402} C_VEL
LIN {X 0,Y 502.912,Z 164.84,A -85,B 0,C 180,E1 -5945.614,E2 -5945.614} C_VEL
LIN {X 0,Y 502.846,Z 164.848,A -85,B 0,C 180,E1 -5948.844,E2 -5948.844} C_VEL
LIN {X 0,Y 502.844,Z 164.852,A -85,B 0,C 180,E1 -5952.102,E2 -5952.102} C_VEL
LIN {X 0,Y 502.847,Z 164.85,A -85,B 0,C 180,E1 -5955.4,E2 -5955.4} C_VEL
LIN {X 0,Y 502.839,Z 164.849,A -85,B 0,C 180,E1 -5958.12,E2 -5958.12} C_VEL
LIN {X 0,Y 502.827,Z 164.853,A -85,B 0,C 180,E1 -5960.536,E2 -5960.536} C_VEL
LIN {X 0,Y 502.785,Z 164.854,A -85,B 0,C 180,E1 -5963.041,E2 -5963.041} C_VEL
LIN {X 0,Y 502.82,Z 164.855,A -85,B 0,C 180,E1 -5965.677,E2 -5965.677} C_VEL
LIN {X 0,Y 502.839,Z 164.848,A -85,B 0,C 180,E1 -5968.373,E2 -5968.373} C_VEL
LIN {X 0,Y 502.791,Z 164.855,A -85,B 0,C 180,E1 -5971.499,E2 -5971.499} C_VEL
LIN {X 0,Y 502.801,Z 164.857,A -85,B 0,C 180,E1 -5973.994,E2 -5973.994} C_VEL
LIN {X 0,Y 502.735,Z 164.862,A -85,B 0,C 180,E1 -5977.172,E2 -5977.172} C_VEL
LIN {X 0,Y 502.786,Z 164.853,A -85,B 0,C 180,E1 -5980.016,E2 -5980.016} C_VEL
LIN {X 0,Y 502.802,Z 164.852,A -85,B 0,C 180,E1 -5982.2,E2 -5982.2} C_VEL
LIN {X 0,Y 502.801,Z 164.853,A -85,B 0,C 180,E1 -5985.469,E2 -5985.469} C_VEL
LIN {X 0,Y 502.819,Z 164.851,A -85,B 0,C 180,E1 -5988.934,E2 -5988.934} C_VEL
LIN {X 0,Y 502.787,Z 164.855,A -85,B 0,C 180,E1 -5992.046,E2 -5992.046} C_VEL
LIN {X 0,Y 502.696,Z 164.867,A -85,B 0,C 180,E1 -5994.182,E2 -5994.182} C_VEL
LIN {X 0,Y 502.665,Z 165.48,A -85,B 0,C 180,E1 -5995.024,E2 -5995.024} C_VEL
LIN {X 0,Y 502.642,Z 168.595,A -85,B 0,C 180,E1 -5997.171,E2 -5997.171} C_VEL
LIN {X 0,Y 501.959,Z 169.639,A -85,B 0,C 180,E1 -5997.829,E2 -5997.829} C_VEL
LIN {X 0,Y 499.084,Z 171.549,A -85,B 0,C 180,E1 -5998.893,E2 -5998.893} C_VEL
LIN {X 0,Y 496.653,Z 173.1,A -85,B 0,C 180,E1 -5999.75,E2 -5999.75} C_VEL
LIN {X 0,Y 495.598,Z 174.206,A -85,B 0,C 180,E1 -6000.413,E2 -6000.413} C_VEL
LIN {X 0,Y 495.507,Z 174.55,A -85,B 0,C 180,E1 -6000.639,E2 -6000.639} C_VEL
LIN {X 0,Y 495.438,Z 178.613,A -85,B 0,C 180,E1 -6003.34,E2 -6003.34} C_VEL
LIN {X 0,Y 495.394,Z 182.222,A -85,B 0,C 180,E1 -6005.707,E2 -6005.707} C_VEL
LIN {X 0,Y 495.291,Z 186.328,A -85,B 0,C 180,E1 -6008.351,E2 -6008.351} C_VEL
LIN {X 0,Y 495.196,Z 190.468,A -85,B 0,C 180,E1 -6010.948,E2 -6010.948} C_VEL
LIN {X 0,Y 495.118,Z 194.661,A -85,B 0,C 180,E1 -6013.508,E2 -6013.508} C_VEL
LIN {X 0,Y 495.13,Z 198.133,A -85,B 0,C 180,E1 -6015.565,E2 -6015.565} C_VEL
LIN {X 0,Y 497.831,Z 212.119,A -85,B 0,C 180,E1 -6016.036,E2 -6016.036} C_VEL
LIN {X 0,Y 497.472,Z 225.307,A -85,B 0,C 180,E1 -6016.572,E2 -6016.572} C_VEL
LIN {X 0,Y 497.157,Z 237.166,A -85,B 0,C 180,E1 -6017.239,E2 -6017.239} C_VEL
LIN {X 0,Y 496.788,Z 248.54,A -85,B 0,C 180,E1 -6018.06,E2 -6018.06} C_VEL
LIN {X 0,Y 496.392,Z 258.784,A -85,B 0,C 180,E1 -6018.981,E2 -6018.981} C_VEL
LIN {X 0,Y 496.036,Z 267.974,A -85,B 0,C 180,E1 -6020.005,E2 -6020.005} C_VEL
LIN {X 0,Y 495.723,Z 276.892,A -85,B 0,C 180,E1 -6021.234,E2 -6021.234} C_VEL
LIN {X 0,Y 495.431,Z 284.073,A -85,B 0,C 180,E1 -6022.46,E2 -6022.46} C_VEL
LIN {X 0,Y 495.292,Z 288.916,A -85,B 0,C 180,E1 -6023.482,E2 -6023.482} C_VEL
LIN {X 0,Y 495.13,Z 293.624,A -85,B 0,C 180,E1 -6024.706,E2 -6024.706} C_VEL
LIN {X 0,Y 495.153,Z 297.225,A -85,B 0,C 180,E1 -6025.931,E2 -6025.931} C_VEL
LIN {X 0,Y 495.083,Z 299.089,A -85,B 0,C 180,E1 -6026.745,E2 -6026.745} C_VEL
LIN {X 0,Y 495.033,Z 300.495,A -85,B 0,C 180,E1 -6027.559,E2 -6027.559} C_VEL
LIN {X 0,Y 494.912,Z 302.112,A -85,B 0,C 180,E1 -6029.187,E2 -6029.187} C_VEL
LIN {X 0,Y 494.901,Z 302.348,A -85,B 0,C 180,E1 -6030,E2 -6030} C_VEL
LIN {X 0,Y 494.912,Z 302.164,A -85,B 0,C 180,E1 -6030.814,E2 -6030.814} C_VEL
LIN {X 0,Y 495.033,Z 300.614,A -85,B 0,C 180,E1 -6032.441,E2 -6032.441} C_VEL
LIN {X 0,Y 495.083,Z 299.26,A -85,B 0,C 180,E1 -6033.255,E2 -6033.255} C_VEL
LIN {X 0,Y 495.122,Z 296.4,A -85,B 0,C 180,E1 -6034.478,E2 -6034.478} C_VEL
LIN {X 0,Y 495.248,Z 292.518,A -85,B 0,C 180,E1 -6035.701,E2 -6035.701} C_VEL
LIN {X 0,Y 495.309,Z 287.515,A -85,B 0,C 180,E1 -6036.927,E2 -6036.927} C_VEL
LIN {X 0,Y 495.536,Z 281.211,A -85,B 0,C 180,E1 -6038.154,E2 -6038.154} C_VEL
LIN {X 0,Y 495.817,Z 273.319,A -85,B 0,C 180,E1 -6039.382,E2 -6039.382} C_VEL
LIN {X 0,Y 496.172,Z 265.272,A -85,B 0,C 180,E1 -6040.405,E2 -6040.405} C_VEL
LIN {X 0,Y 496.501,Z 255.453,A -85,B 0,C 180,E1 -6041.43,E2 -6041.43} C_VEL
LIN {X 0,Y 496.887,Z 244.551,A -85,B 0,C 180,E1 -6042.343,E2 -6042.343} C_VEL
LIN {X 0,Y 497.226,Z 233.592,A -85,B 0,C 180,E1 -6043.071,E2 -6043.071} C_VEL
LIN {X 0,Y 497.6,Z 221.639,A -85,B 0,C 180,E1 -6043.685,E2 -6043.685} C_VEL
LIN {X 0,Y 497.657,Z 210.951,A -85,B 0,C 180,E1 -6044.1,E2 -6044.1} C_VEL
LIN {X 0,Y 495.114,Z 198.108,A -85,B 0,C 180,E1 -6044.541,E2 -6044.541} C_VEL
LIN {X 0,Y 495.193,Z 192.293,A -85,B 0,C 180,E1 -6048.029,E2 -6048.029} C_VEL
LIN {X 0,Y 495.242,Z 187.842,A -85,B 0,C 180,E1 -6050.78,E2 -6050.78} C_VEL
LIN {X 0,Y 495.321,Z 183.742,A -85,B 0,C 180,E1 -6053.409,E2 -6053.409} C_VEL
LIN {X 0,Y 495.396,Z 181.002,A -85,B 0,C 180,E1 -6055.189,E2 -6055.189} C_VEL
LIN {X 0,Y 495.511,Z 176.079,A -85,B 0,C 180,E1 -6058.433,E2 -6058.433} C_VEL
LIN {X 0,Y 495.565,Z 171.308,A -85,B 0,C 180,E1 -6061.65,E2 -6061.65} C_VEL
LIN {X 0,Y 495.686,Z 166.92,A -85,B 0,C 180,E1 -6064.679,E2 -6064.679} C_VEL
LIN {X 0,Y 495.641,Z 165.749,A -85,B 0,C 180,E1 -6065.547,E2 -6065.547} C_VEL
LIN {X 0,Y 495.736,Z 165.736,A -85,B 0,C 180,E1 -6068.764,E2 -6068.764} C_VEL
LIN {X 0,Y 495.745,Z 165.735,A -85,B 0,C 180,E1 -6071.782,E2 -6071.782} C_VEL
LIN {X 0,Y 495.739,Z 165.734,A -85,B 0,C 180,E1 -6075.141,E2 -6075.141} C_VEL
LIN {X 0,Y 495.758,Z 165.729,A -85,B 0,C 180,E1 -6078.219,E2 -6078.219} C_VEL
LIN {X 0,Y 495.746,Z 165.732,A -85,B 0,C 180,E1 -6081.234,E2 -6081.234} C_VEL
LIN {X 0,Y 495.735,Z 165.736,A -85,B 0,C 180,E1 -6084.461,E2 -6084.461} C_VEL
LIN {X 0,Y 495.767,Z 165.731,A -85,B 0,C 180,E1 -6087.405,E2 -6087.405} C_VEL
LIN {X 0,Y 495.768,Z 165.729,A -85,B 0,C 180,E1 -6090.254,E2 -6090.254} C_VEL
LIN {X 0,Y 495.825,Z 165.721,A -85,B 0,C 180,E1 -6093.251,E2 -6093.251} C_VEL
LIN {X 0,Y 495.743,Z 165.732,A -85,B 0,C 180,E1 -6096.612,E2 -6096.612} C_VEL
LIN {X 0,Y 495.78,Z 165.729,A -85,B 0,C 180,E1 -6099.324,E2 -6099.324} C_VEL
LIN {X 0,Y 495.782,Z 165.728,A -85,B 0,C 180,E1 -6101.828,E2 -6101.828} C_VEL
LIN {X 0,Y 495.825,Z 165.725,A -85,B 0,C 180,E1 -6104.548,E2 -6104.548} C_VEL
LIN {X 0,Y 495.829,Z 165.726,A -85,B 0,C 180,E1 -6107.965,E2 -6107.965} C_VEL
LIN {X 0,Y 495.807,Z 165.723,A -85,B 0,C 180,E1 -6111.03,E2 -6111.03} C_VEL
LIN {X 0,Y 495.819,Z 165.725,A -85,B 0,C 180,E1 -6113.489,E2 -6113.489} C_VEL
LIN {X 0,Y 495.836,Z 165.724,A -85,B 0,C 180,E1 -6116.75,E2 -6116.75} C_VEL
LIN {X 0,Y 496.006,Z 165.7,A -85,B 0,C 180,E1 -6119.188,E2 -6119.188} C_VEL
LIN {X 0,Y 495.872,Z 165.72,A -85,B 0,C 180,E1 -6121.624,E2 -6121.624} C_VEL
LIN {X 0,Y 495.839,Z 165.724,A -85,B 0,C 180,E1 -6123.25,E2 -6123.25} C_VEL
LIN {X 0,Y 495.821,Z 165.723,A -85,B 0,C 180,E1 -6126.511,E2 -6126.511} C_VEL
LIN {X 0,Y 495.805,Z 165.726,A -85,B 0,C 180,E1 -6128.97,E2 -6128.97} C_VEL
LIN {X 0,Y 495.853,Z 165.722,A -85,B 0,C 180,E1 -6132.275,E2 -6132.275} C_VEL
LIN {X 0,Y 495.808,Z 165.726,A -85,B 0,C 180,E1 -6135.624,E2 -6135.624} C_VEL
LIN {X 0,Y 495.783,Z 165.729,A -85,B 0,C 180,E1 -6139.029,E2 -6139.029} C_VEL
LIN {X 0,Y 495.743,Z 165.731,A -85,B 0,C 180,E1 -6141.629,E2 -6141.629} C_VEL
LIN {X 0,Y 495.751,Z 165.73,A -85,B 0,C 180,E1 -6144.866,E2 -6144.866} C_VEL
LIN {X 0,Y 495.814,Z 165.724,A -85,B 0,C 180,E1 -6146.974,E2 -6146.974} C_VEL
LIN {X 0,Y 495.766,Z 165.73,A -85,B 0,C 180,E1 -6150.147,E2 -6150.147} C_VEL
LIN {X 0,Y 495.794,Z 165.726,A -85,B 0,C 180,E1 -6153.244,E2 -6153.244} C_VEL
LIN {X 0,Y 495.694,Z 165.741,A -85,B 0,C 180,E1 -6156.084,E2 -6156.084} C_VEL
LIN {X 0,Y 495.74,Z 165.731,A -85,B 0,C 180,E1 -6158.765,E2 -6158.765} C_VEL
LIN {X 0,Y 495.757,Z 165.73,A -85,B 0,C 180,E1 -6161.781,E2 -6161.781} C_VEL
LIN {X 0,Y 495.738,Z 165.734,A -85,B 0,C 180,E1 -6165.141,E2 -6165.141} C_VEL
LIN {X 0,Y 495.757,Z 165.735,A -85,B 0,C 180,E1 -6168.219,E2 -6168.219} C_VEL
LIN {X 0,Y 495.778,Z 165.733,A -85,B 0,C 180,E1 -6171.541,E2 -6171.541} C_VEL
LIN {X 0,Y 496.062,Z 167.523,A -85,B 0,C 180,E1 -6172.503,E2 -6172.503} C_VEL
LIN {X 0,Y 496.601,Z 171.931,A -85,B 0,C 180,E1 -6174.533,E2 -6174.533} C_VEL
LIN {X 0,Y 496.433,Z 178.714,A -85,B 0,C 180,E1 -6177.455,E2 -6177.455} C_VEL
LIN {X 0,Y 496.189,Z 186.632,A -85,B 0,C 180,E1 -6180.748,E2 -6180.748} C_VEL
LIN {X 0,Y 495.987,Z 192.74,A -85,B 0,C 180,E1 -6183.214,E2 -6183.214} C_VEL
LIN {X 0,Y 495.807,Z 200.24,A -85,B 0,C 180,E1 -6186.172,E2 -6186.172} C_VEL
LIN {X 0,Y 495.619,Z 208.143,A -85,B 0,C 180,E1 -6189.237,E2 -6189.237} C_VEL
LIN {X 0,Y 495.462,Z 216.009,A -85,B 0,C 180,E1 -6192.272,E2 -6192.272} C_VEL
LIN {X 0,Y 495.308,Z 224.491,A -85,B 0,C 180,E1 -6195.491,E2 -6195.491} C_VEL
LIN {X 0,Y 497.636,Z 238.308,A -85,B 0,C 180,E1 -6195.913,E2 -6195.913} C_VEL
LIN {X 0,Y 497.484,Z 251.237,A -85,B 0,C 180,E1 -6196.416,E2 -6196.416} C_VEL
LIN {X 0,Y 497.098,Z 262.748,A -85,B 0,C 180,E1 -6197.019,E2 -6197.019} C_VEL
LIN {X 0,Y 496.742,Z 273.587,A -85,B 0,C 180,E1 -6197.747,E2 -6197.747} C_VEL
LIN {X 0,Y 496.399,Z 284.467,A -85,B 0,C 180,E1 -6198.671,E2 -6198.671} C_VEL
LIN {X 0,Y 495.995,Z 293.332,A -85,B 0,C 180,E1 -6199.592,E2 -6199.592} C_VEL
LIN {X 0,Y 495.673,Z 302.959,A -85,B 0,C 180,E1 -6200.821,E2 -6200.821} C_VEL
LIN {X 0,Y 495.404,Z 310.621,A -85,B 0,C 180,E1 -6202.049,E2 -6202.049} C_VEL
LIN {X 0,Y 495.204,Z 317.679,A -85,B 0,C 180,E1 -6203.481,E2 -6203.481} C_VEL
LIN {X 0,Y 495.123,Z 322.372,A -85,B 0,C 180,E1 -6204.706,E2 -6204.706} C_VEL
LIN {X 0,Y 495.049,Z 325.958,A -85,B 0,C 180,E1 -6205.929,E2 -6205.929} C_VEL
LIN {X 0,Y 495.043,Z 327.807,A -85,B 0,C 180,E1 -6206.744,E2 -6206.744} C_VEL
LIN {X 0,Y 494.961,Z 330.183,A -85,B 0,C 180,E1 -6208.372,E2 -6208.372} C_VEL
LIN {X 0,Y 494.898,Z 331,A -85,B 0,C 180,E1 -6210,E2 -6210} C_VEL
LIN {X 0,Y 494.961,Z 330.185,A -85,B 0,C 180,E1 -6211.627,E2 -6211.627} C_VEL
LIN {X 0,Y 495.043,Z 327.81,A -85,B 0,C 180,E1 -6213.255,E2 -6213.255} C_VEL
LIN {X 0,Y 495.029,Z 324.896,A -85,B 0,C 180,E1 -6214.478,E2 -6214.478} C_VEL
LIN {X 0,Y 495.21,Z 319.803,A -85,B 0,C 180,E1 -6215.999,E2 -6215.999} C_VEL
LIN {X 0,Y 495.277,Z 313.87,A -85,B 0,C 180,E1 -6217.337,E2 -6217.337} C_VEL
LIN {X 0,Y 495.557,Z 307.004,A -85,B 0,C 180,E1 -6218.564,E2 -6218.564} C_VEL
LIN {X 0,Y 495.85,Z 298.415,A -85,B 0,C 180,E1 -6219.792,E2 -6219.792} C_VEL
LIN {X 0,Y 496.174,Z 289.601,A -85,B 0,C 180,E1 -6220.817,E2 -6220.817} C_VEL
LIN {X 0,Y 496.58,Z 278.747,A -85,B 0,C 180,E1 -6221.842,E2 -6221.842} C_VEL
LIN {X 0,Y 496.872,Z 268.215,A -85,B 0,C 180,E1 -6222.636,E2 -6222.636} C_VEL
LIN {X 0,Y 497.286,Z 255.505,A -85,B 0,C 180,E1 -6223.381,E2 -6223.381} C_VEL
LIN {X 0,Y 497.714,Z 242.499,A -85,B 0,C 180,E1 -6223.941,E2 -6223.941} C_VEL
LIN {X 0,Y 497.437,Z 237.096,A -85,B 0,C 180,E1 -6224.132,E2 -6224.132} C_VEL
LIN {X 0,Y 495.307,Z 224.492,A -85,B 0,C 180,E1 -6224.508,E2 -6224.508} C_VEL
LIN {X 0,Y 495.461,Z 216.01,A -85,B 0,C 180,E1 -6227.728,E2 -6227.728} C_VEL
LIN {X 0,Y 495.64,Z 208.144,A -85,B 0,C 180,E1 -6230.762,E2 -6230.762} C_VEL
LIN {X 0,Y 495.808,Z 200.229,A -85,B 0,C 180,E1 -6233.827,E2 -6233.827} C_VEL
LIN {X 0,Y 496.018,Z 192.3,A -85,B 0,C 180,E1 -6236.962,E2 -6236.962} C_VEL
LIN {X 0,Y 496.283,Z 184.187,A -85,B 0,C 180,E1 -6240.249,E2 -6240.249} C_VEL
LIN {X 0,Y 496.486,Z 176.785,A -85,B 0,C 180,E1 -6243.366,E2 -6243.366} C_VEL
LIN {X 0,Y 496.608,Z 171.931,A -85,B 0,C 180,E1 -6245.466,E2 -6245.466} C_VEL
LIN {X 0,Y 496.079,Z 167.444,A -85,B 0,C 180,E1 -6247.53,E2 -6247.53} C_VEL
LIN {X 0,Y 495.776,Z 165.733,A -85,B 0,C 180,E1 -6248.459,E2 -6248.459} C_VEL
LIN {X 0,Y 495.756,Z 165.735,A -85,B 0,C 180,E1 -6251.781,E2 -6251.781} C_VEL
LIN {X 0,Y 495.736,Z 165.736,A -85,B 0,C 180,E1 -6255.14,E2 -6255.14} C_VEL
LIN {X 0,Y 495.755,Z 165.731,A -85,B 0,C 180,E1 -6258.219,E2 -6258.219} C_VEL
LIN {X 0,Y 495.742,Z 165.73,A -85,B 0,C 180,E1 -6261.234,E2 -6261.234} C_VEL
LIN {X 0,Y 495.735,Z 165.734,A -85,B 0,C 180,E1 -6264.461,E2 -6264.461} C_VEL
LIN {X 0,Y 495.766,Z 165.731,A -85,B 0,C 180,E1 -6267.405,E2 -6267.405} C_VEL
LIN {X 0,Y 495.765,Z 165.731,A -85,B 0,C 180,E1 -6270.253,E2 -6270.253} C_VEL
LIN {X 0,Y 495.822,Z 165.722,A -85,B 0,C 180,E1 -6273.251,E2 -6273.251} C_VEL
LIN {X 0,Y 495.74,Z 165.731,A -85,B 0,C 180,E1 -6276.612,E2 -6276.612} C_VEL
LIN {X 0,Y 495.776,Z 165.73,A -85,B 0,C 180,E1 -6279.324,E2 -6279.324} C_VEL
LIN {X 0,Y 495.791,Z 165.727,A -85,B 0,C 180,E1 -6281.829,E2 -6281.829} C_VEL
LIN {X 0,Y 495.822,Z 165.724,A -85,B 0,C 180,E1 -6284.548,E2 -6284.548} C_VEL
LIN {X 0,Y 495.826,Z 165.724,A -85,B 0,C 180,E1 -6287.965,E2 -6287.965} C_VEL
LIN {X 0,Y 495.804,Z 165.726,A -85,B 0,C 180,E1 -6291.03,E2 -6291.03} C_VEL
LIN {X 0,Y 495.868,Z 165.716,A -85,B 0,C 180,E1 -6294.306,E2 -6294.306} C_VEL
LIN {X 0,Y 495.99,Z 165.702,A -85,B 0,C 180,E1 -6297.564,E2 -6297.564} C_VEL
LIN {X 0,Y 495.997,Z 165.703,A -85,B 0,C 180,E1 -6300,E2 -6300} C_VEL
LIN {X 0,Y 495.989,Z 165.702,A -85,B 0,C 180,E1 -6302.436,E2 -6302.436} C_VEL
LIN {X 0,Y 495.867,Z 165.717,A -85,B 0,C 180,E1 -6305.694,E2 -6305.694} C_VEL
LIN {X 0,Y 495.804,Z 165.724,A -85,B 0,C 180,E1 -6308.97,E2 -6308.97} C_VEL
LIN {X 0,Y 495.826,Z 165.726,A -85,B 0,C 180,E1 -6312.035,E2 -6312.035} C_VEL
LIN {X 0,Y 495.822,Z 165.725,A -85,B 0,C 180,E1 -6315.452,E2 -6315.452} C_VEL
LIN {X 0,Y 495.805,Z 165.726,A -85,B 0,C 180,E1 -6318.248,E2 -6318.248} C_VEL
LIN {X 0,Y 495.772,Z 165.73,A -85,B 0,C 180,E1 -6320.757,E2 -6320.757} C_VEL
LIN {X 0,Y 495.74,Z 165.732,A -85,B 0,C 180,E1 -6323.388,E2 -6323.388} C_VEL
LIN {X 0,Y 495.822,Z 165.721,A -85,B 0,C 180,E1 -6326.75,E2 -6326.75} C_VEL
LIN {X 0,Y 495.765,Z 165.73,A -85,B 0,C 180,E1 -6329.747,E2 -6329.747} C_VEL
LIN {X 0,Y 495.766,Z 165.731,A -85,B 0,C 180,E1 -6332.595,E2 -6332.595} C_VEL
LIN {X 0,Y 495.735,Z 165.735,A -85,B 0,C 180,E1 -6335.539,E2 -6335.539} C_VEL
LIN {X 0,Y 495.743,Z 165.732,A -85,B 0,C 180,E1 -6338.766,E2 -6338.766} C_VEL
LIN {X 0,Y 495.755,Z 165.729,A -85,B 0,C 180,E1 -6341.782,E2 -6341.782} C_VEL
LIN {X 0,Y 495.749,Z 165.732,A -85,B 0,C 180,E1 -6345.14,E2 -6345.14} C_VEL
LIN {X 0,Y 495.756,Z 165.734,A -85,B 0,C 180,E1 -6348.219,E2 -6348.219} C_VEL
LIN {X 0,Y 495.744,Z 165.734,A -85,B 0,C 180,E1 -6351.408,E2 -6351.408} C_VEL
LIN {X 0,Y 495.608,Z 165.752,A -85,B 0,C 180,E1 -6354.451,E2 -6354.451} C_VEL
LIN {X 0,Y 495.601,Z 168.921,A -85,B 0,C 180,E1 -6356.79,E2 -6356.79} C_VEL
LIN {X 0,Y 495.541,Z 173.446,A -85,B 0,C 180,E1 -6359.898,E2 -6359.898} C_VEL
LIN {X 0,Y 495.507,Z 174.55,A -85,B 0,C 180,E1 -6360.639,E2 -6360.639} C_VEL
LIN {X 0,Y 494.813,Z 175.622,A -85,B 0,C 180,E1 -6361.306,E2 -6361.306} C_VEL
LIN {X 0,Y 491.907,Z 177.555,A -85,B 0,C 180,E1 -6362.384,E2 -6362.384} C_VEL
LIN {X 0,Y 489.457,Z 179.118,A -85,B 0,C 180,E1 -6363.252,E2 -6363.252} C_VEL
LIN {X 0,Y 488.405,Z 180.234,A -85,B 0,C 180,E1 -6363.925,E2 -6363.925} C_VEL
LIN {X 0,Y 488.318,Z 180.585,A -85,B 0,C 180,E1 -6364.154,E2 -6364.154} C_VEL
LIN {X 0,Y 488.298,Z 183.737,A -85,B 0,C 180,E1 -6366.234,E2 -6366.234} C_VEL
LIN {X 0,Y 488.202,Z 188.544,A -85,B 0,C 180,E1 -6369.345,E2 -6369.345} C_VEL
LIN {X 0,Y 488.1,Z 193.438,A -85,B 0,C 180,E1 -6372.4,E2 -6372.4} C_VEL
LIN {X 0,Y 488.034,Z 198.331,A -85,B 0,C 180,E1 -6375.35,E2 -6375.35} C_VEL
LIN {X 0,Y 490.837,Z 212.35,A -85,B 0,C 180,E1 -6375.833,E2 -6375.833} C_VEL
LIN {X 0,Y 490.619,Z 224.42,A -85,B 0,C 180,E1 -6376.329,E2 -6376.329} C_VEL
LIN {X 0,Y 490.253,Z 235.147,A -85,B 0,C 180,E1 -6376.911,E2 -6376.911} C_VEL
LIN {X 0,Y 489.912,Z 246.188,A -85,B 0,C 180,E1 -6377.679,E2 -6377.679} C_VEL
LIN {X 0,Y 489.488,Z 256.877,A -85,B 0,C 180,E1 -6378.614,E2 -6378.614} C_VEL
LIN {X 0,Y 489.149,Z 266.493,A -85,B 0,C 180,E1 -6379.654,E2 -6379.654} C_VEL
LIN {X 0,Y 488.82,Z 274.369,A -85,B 0,C 180,E1 -6380.692,E2 -6380.692} C_VEL
LIN {X 0,Y 488.473,Z 282.07,A -85,B 0,C 180,E1 -6381.936,E2 -6381.936} C_VEL
LIN {X 0,Y 488.222,Z 289.132,A -85,B 0,C 180,E1 -6383.387,E2 -6383.387} C_VEL
LIN {X 0,Y 488.076,Z 293.838,A -85,B 0,C 180,E1 -6384.63,E2 -6384.63} C_VEL
LIN {X 0,Y 488.072,Z 297.439,A -85,B 0,C 180,E1 -6385.871,E2 -6385.871} C_VEL
LIN {X 0,Y 488.008,Z 299.303,A -85,B 0,C 180,E1 -6386.698,E2 -6386.698} C_VEL
LIN {X 0,Y 487.942,Z 300.708,A -85,B 0,C 180,E1 -6387.524,E2 -6387.524} C_VEL
LIN {X 0,Y 487.836,Z 302.324,A -85,B 0,C 180,E1 -6389.175,E2 -6389.175} C_VEL
LIN {X 0,Y 487.822,Z 302.561,A -85,B 0,C 180,E1 -6390,E2 -6390} C_VEL
LIN {X 0,Y 487.835,Z 302.376,A -85,B 0,C 180,E1 -6390.826,E2 -6390.826} C_VEL
LIN {X 0,Y 487.942,Z 300.826,A -85,B 0,C 180,E1 -6392.477,E2 -6392.477} C_VEL
LIN {X 0,Y 488.009,Z 299.472,A -85,B 0,C 180,E1 -6393.303,E2 -6393.303} C_VEL
LIN {X 0,Y 488.02,Z 296.612,A -85,B 0,C 180,E1 -6394.543,E2 -6394.543} C_VEL
LIN {X 0,Y 488.197,Z 292.729,A -85,B 0,C 180,E1 -6395.784,E2 -6395.784} C_VEL
LIN {X 0,Y 488.258,Z 287.726,A -85,B 0,C 180,E1 -6397.027,E2 -6397.027} C_VEL
LIN {X 0,Y 488.508,Z 281.421,A -85,B 0,C 180,E1 -6398.272,E2 -6398.272} C_VEL
LIN {X 0,Y 488.815,Z 273.528,A -85,B 0,C 180,E1 -6399.517,E2 -6399.517} C_VEL
LIN {X 0,Y 489.158,Z 265.481,A -85,B 0,C 180,E1 -6400.556,E2 -6400.556} C_VEL
LIN {X 0,Y 489.554,Z 255.661,A -85,B 0,C 180,E1 -6401.595,E2 -6401.595} C_VEL
LIN {X 0,Y 489.926,Z 245.999,A -85,B 0,C 180,E1 -6402.426,E2 -6402.426} C_VEL
LIN {X 0,Y 490.239,Z 235.27,A -85,B 0,C 180,E1 -6403.172,E2 -6403.172} C_VEL
LIN {X 0,Y 490.671,Z 222.968,A -85,B 0,C 180,E1 -6403.829,E2 -6403.829} C_VEL
LIN {X 0,Y 490.801,Z 211.909,A -85,B 0,C 180,E1 -6404.274,E2 -6404.274} C_VEL
LIN {X 0,Y 488.034,Z 198.303,A -85,B 0,C 180,E1 -6404.757,E2 -6404.757} C_VEL
LIN {X 0,Y 488.111,Z 192.726,A -85,B 0,C 180,E1 -6408.14,E2 -6408.14} C_VEL
LIN {X 0,Y 488.192,Z 188.001,A -85,B 0,C 180,E1 -6411.094,E2 -6411.094} C_VEL
LIN {X 0,Y 488.295,Z 183.892,A -85,B 0,C 180,E1 -6413.766,E2 -6413.766} C_VEL
LIN {X 0,Y 488.349,Z 179.757,A -85,B 0,C 180,E1 -6416.496,E2 -6416.496} C_VEL
LIN {X 0,Y 488.467,Z 175.598,A -85,B 0,C 180,E1 -6419.287,E2 -6419.287} C_VEL
LIN {X 0,Y 488.551,Z 171.412,A -85,B 0,C 180,E1 -6422.158,E2 -6422.158} C_VEL
LIN {X 0,Y 488.617,Z 167.19,A -85,B 0,C 180,E1 -6425.123,E2 -6425.123} C_VEL
LIN {X 0,Y 488.646,Z 166.619,A -85,B 0,C 180,E1 -6426.348,E2 -6426.348} C_VEL
LIN {X 0,Y 488.685,Z 166.613,A -85,B 0,C 180,E1 -6429.256,E2 -6429.256} C_VEL
LIN {X 0,Y 488.672,Z 166.615,A -85,B 0,C 180,E1 -6432.528,E2 -6432.528} C_VEL
LIN {X 0,Y 488.703,Z 166.612,A -85,B 0,C 180,E1 -6435.197,E2 -6435.197} C_VEL
LIN {X 0,Y 488.708,Z 166.607,A -85,B 0,C 180,E1 -6438.4,E2 -6438.4} C_VEL
LIN {X 0,Y 488.694,Z 166.613,A -85,B 0,C 180,E1 -6440.949,E2 -6440.949} C_VEL
LIN {X 0,Y 488.653,Z 166.616,A -85,B 0,C 180,E1 -6443.866,E2 -6443.866} C_VEL
LIN {X 0,Y 488.736,Z 166.606,A -85,B 0,C 180,E1 -6446.877,E2 -6446.877} C_VEL
LIN {X 0,Y 488.725,Z 166.608,A -85,B 0,C 180,E1 -6449.781,E2 -6449.781} C_VEL
LIN {X 0,Y 488.793,Z 166.598,A -85,B 0,C 180,E1 -6453.056,E2 -6453.056} C_VEL
LIN {X 0,Y 488.681,Z 166.615,A -85,B 0,C 180,E1 -6456.254,E2 -6456.254} C_VEL
LIN {X 0,Y 488.748,Z 166.604,A -85,B 0,C 180,E1 -6459.176,E2 -6459.176} C_VEL
LIN {X 0,Y 488.75,Z 166.606,A -85,B 0,C 180,E1 -6461.631,E2 -6461.631} C_VEL
LIN {X 0,Y 488.763,Z 166.603,A -85,B 0,C 180,E1 -6465,E2 -6465} C_VEL
LIN {X 0,Y 488.806,Z 166.597,A -85,B 0,C 180,E1 -6468.387,E2 -6468.387} C_VEL
LIN {X 0,Y 488.762,Z 166.604,A -85,B 0,C 180,E1 -6471.733,E2 -6471.733} C_VEL
LIN {X 0,Y 488.825,Z 166.594,A -85,B 0,C 180,E1 -6474.224,E2 -6474.224} C_VEL
LIN {X 0,Y 488.958,Z 166.578,A -85,B 0,C 180,E1 -6477.529,E2 -6477.529} C_VEL
LIN {X 0,Y 488.971,Z 166.578,A -85,B 0,C 180,E1 -6480,E2 -6480} C_VEL
LIN {X 0,Y 488.96,Z 166.577,A -85,B 0,C 180,E1 -6482.471,E2 -6482.471} C_VEL
LIN {X 0,Y 488.828,Z 166.592,A -85,B 0,C 180,E1 -6485.776,E2 -6485.776} C_VEL
LIN {X 0,Y 488.761,Z 166.602,A -85,B 0,C 180,E1 -6488.267,E2 -6488.267} C_VEL
LIN {X 0,Y 488.832,Z 166.594,A -85,B 0,C 180,E1 -6491.612,E2 -6491.612} C_VEL
LIN {X 0,Y 488.763,Z 166.604,A -85,B 0,C 180,E1 -6495,E2 -6495} C_VEL
LIN {X 0,Y 488.748,Z 166.605,A -85,B 0,C 180,E1 -6498.442,E2 -6498.442} C_VEL
LIN {X 0,Y 488.708,Z 166.608,A -85,B 0,C 180,E1 -6501.071,E2 -6501.071} C_VEL
LIN {X 0,Y 488.677,Z 166.613,A -85,B 0,C 180,E1 -6503.746,E2 -6503.746} C_VEL
LIN {X 0,Y 488.793,Z 166.599,A -85,B 0,C 180,E1 -6506.944,E2 -6506.944} C_VEL
LIN {X 0,Y 488.711,Z 166.61,A -85,B 0,C 180,E1 -6510.363,E2 -6510.363} C_VEL
LIN {X 0,Y 488.735,Z 166.605,A -85,B 0,C 180,E1 -6513.484,E2 -6513.484} C_VEL
LIN {X 0,Y 488.653,Z 166.616,A -85,B 0,C 180,E1 -6516.35,E2 -6516.35} C_VEL
LIN {X 0,Y 488.69,Z 166.613,A -85,B 0,C 180,E1 -6519.255,E2 -6519.255} C_VEL
LIN {X 0,Y 488.708,Z 166.609,A -85,B 0,C 180,E1 -6521.6,E2 -6521.6} C_VEL
LIN {X 0,Y 488.703,Z 166.613,A -85,B 0,C 180,E1 -6524.803,E2 -6524.803} C_VEL
LIN {X 0,Y 488.693,Z 166.611,A -85,B 0,C 180,E1 -6527.475,E2 -6527.475} C_VEL
LIN {X 0,Y 488.735,Z 166.61,A -85,B 0,C 180,E1 -6529.677,E2 -6529.677} C_VEL
LIN {X 0,Y 488.76,Z 166.823,A -85,B 0,C 180,E1 -6531.545,E2 -6531.545} C_VEL
LIN {X 0,Y 489.496,Z 171.847,A -85,B 0,C 180,E1 -6533.938,E2 -6533.938} C_VEL
LIN {X 0,Y 489.552,Z 176.352,A -85,B 0,C 180,E1 -6535.952,E2 -6535.952} C_VEL
LIN {X 0,Y 489.273,Z 183.116,A -85,B 0,C 180,E1 -6538.861,E2 -6538.861} C_VEL
LIN {X 0,Y 489.074,Z 189.929,A -85,B 0,C 180,E1 -6541.692,E2 -6541.692} C_VEL
LIN {X 0,Y 488.852,Z 197.857,A -85,B 0,C 180,E1 -6544.921,E2 -6544.921} C_VEL
LIN {X 0,Y 488.644,Z 205.798,A -85,B 0,C 180,E1 -6548.041,E2 -6548.041} C_VEL
LIN {X 0,Y 488.49,Z 213.709,A -85,B 0,C 180,E1 -6551.112,E2 -6551.112} C_VEL
LIN {X 0,Y 488.29,Z 222.862,A -85,B 0,C 180,E1 -6554.653,E2 -6554.653} C_VEL
LIN {X 0,Y 488.235,Z 224.491,A -85,B 0,C 180,E1 -6555.276,E2 -6555.276} C_VEL
LIN {X 0,Y 490.605,Z 238.307,A -85,B 0,C 180,E1 -6555.707,E2 -6555.707} C_VEL
LIN {X 0,Y 490.812,Z 242.497,A -85,B 0,C 180,E1 -6555.858,E2 -6555.858} C_VEL
LIN {X 0,Y 490.492,Z 254.508,A -85,B 0,C 180,E1 -6556.377,E2 -6556.377} C_VEL
LIN {X 0,Y 490.048,Z 266.062,A -85,B 0,C 180,E1 -6557.041,E2 -6557.041} C_VEL
LIN {X 0,Y 489.714,Z 276.192,A -85,B 0,C 180,E1 -6557.779,E2 -6557.779} C_VEL
LIN {X 0,Y 489.332,Z 286.604,A -85,B 0,C 180,E1 -6558.715,E2 -6558.715} C_VEL
LIN {X 0,Y 488.945,Z 295.112,A -85,B 0,C 180,E1 -6559.649,E2 -6559.649} C_VEL
LIN {X 0,Y 488.657,Z 302.959,A -85,B 0,C 180,E1 -6560.688,E2 -6560.688} C_VEL
LIN {X 0,Y 488.361,Z 310.621,A -85,B 0,C 180,E1 -6561.934,E2 -6561.934} C_VEL
LIN {X 0,Y 488.141,Z 317.679,A -85,B 0,C 180,E1 -6563.386,E2 -6563.386} C_VEL
LIN {X 0,Y 488.06,Z 322.372,A -85,B 0,C 180,E1 -6564.629,E2 -6564.629} C_VEL
LIN {X 0,Y 487.947,Z 325.958,A -85,B 0,C 180,E1 -6565.87,E2 -6565.87} C_VEL
LIN {X 0,Y 487.967,Z 327.807,A -85,B 0,C 180,E1 -6566.697,E2 -6566.697} C_VEL
LIN {X 0,Y 487.889,Z 330.183,A -85,B 0,C 180,E1 -6568.349,E2 -6568.349} C_VEL
LIN {X 0,Y 487.819,Z 331,A -85,B 0,C 180,E1 -6570,E2 -6570} C_VEL
LIN {X 0,Y 487.889,Z 330.184,A -85,B 0,C 180,E1 -6571.651,E2 -6571.651} C_VEL
LIN {X 0,Y 487.966,Z 327.81,A -85,B 0,C 180,E1 -6573.302,E2 -6573.302} C_VEL
LIN {X 0,Y 487.938,Z 324.896,A -85,B 0,C 180,E1 -6574.543,E2 -6574.543} C_VEL
LIN {X 0,Y 488.105,Z 320.949,A -85,B 0,C 180,E1 -6575.784,E2 -6575.784} C_VEL
LIN {X 0,Y 488.19,Z 314.877,A -85,B 0,C 180,E1 -6577.236,E2 -6577.236} C_VEL
LIN {X 0,Y 488.454,Z 308.237,A -85,B 0,C 180,E1 -6578.481,E2 -6578.481} C_VEL
LIN {X 0,Y 488.763,Z 299.993,A -85,B 0,C 180,E1 -6579.727,E2 -6579.727} C_VEL
LIN {X 0,Y 489.069,Z 291.542,A -85,B 0,C 180,E1 -6580.767,E2 -6580.767} C_VEL
LIN {X 0,Y 489.523,Z 281.095,A -85,B 0,C 180,E1 -6581.805,E2 -6581.805} C_VEL
LIN {X 0,Y 489.892,Z 269.889,A -85,B 0,C 180,E1 -6582.701,E2 -6582.701} C_VEL
LIN {X 0,Y 490.263,Z 259.409,A -85,B 0,C 180,E1 -6583.365,E2 -6583.365} C_VEL
LIN {X 0,Y 490.686,Z 247.77,A -85,B 0,C 180,E1 -6583.934,E2 -6583.934} C_VEL
LIN {X 0,Y 490.651,Z 238.692,A -85,B 0,C 180,E1 -6584.278,E2 -6584.278} C_VEL
LIN {X 0,Y 488.379,Z 225.622,A -85,B 0,C 180,E1 -6584.692,E2 -6584.692} C_VEL
LIN {X 0,Y 488.238,Z 224.423,A -85,B 0,C 180,E1 -6584.75,E2 -6584.75} C_VEL
LIN {X 0,Y 488.386,Z 217.049,A -85,B 0,C 180,E1 -6587.589,E2 -6587.589} C_VEL
LIN {X 0,Y 488.54,Z 210.345,A -85,B 0,C 180,E1 -6590.197,E2 -6590.197} C_VEL
LIN {X 0,Y 488.733,Z 203.045,A -85,B 0,C 180,E1 -6593.026,E2 -6593.026} C_VEL
LIN {X 0,Y 488.894,Z 195.565,A -85,B 0,C 180,E1 -6596.004,E2 -6596.004} C_VEL
LIN {X 0,Y 489.109,Z 188.798,A -85,B 0,C 180,E1 -6598.776,E2 -6598.776} C_VEL
LIN {X 0,Y 489.358,Z 182.015,A -85,B 0,C 180,E1 -6601.604,E2 -6601.604} C_VEL
LIN {X 0,Y 489.573,Z 175.222,A -85,B 0,C 180,E1 -6604.543,E2 -6604.543} C_VEL
LIN {X 0,Y 489.441,Z 170.945,A -85,B 0,C 180,E1 -6606.475,E2 -6606.475} C_VEL
LIN {X 0,Y 488.717,Z 166.612,A -85,B 0,C 180,E1 -6608.59,E2 -6608.59} C_VEL
LIN {X 0,Y 488.706,Z 166.612,A -85,B 0,C 180,E1 -6611.599,E2 -6611.599} C_VEL
LIN {X 0,Y 488.7,Z 166.61,A -85,B 0,C 180,E1 -6614.802,E2 -6614.802} C_VEL
LIN {X 0,Y 488.69,Z 166.611,A -85,B 0,C 180,E1 -6617.474,E2 -6617.474} C_VEL
LIN {X 0,Y 488.732,Z 166.604,A -85,B 0,C 180,E1 -6619.676,E2 -6619.676} C_VEL
LIN {X 0,Y 488.649,Z 166.616,A -85,B 0,C 180,E1 -6622.838,E2 -6622.838} C_VEL
LIN {X 0,Y 488.726,Z 166.61,A -85,B 0,C 180,E1 -6625.887,E2 -6625.887} C_VEL
LIN {X 0,Y 488.691,Z 166.613,A -85,B 0,C 180,E1 -6628.82,E2 -6628.82} C_VEL
LIN {X 0,Y 488.743,Z 166.604,A -85,B 0,C 180,E1 -6631.671,E2 -6631.671} C_VEL
LIN {X 0,Y 488.725,Z 166.608,A -85,B 0,C 180,E1 -6634.443,E2 -6634.443} C_VEL
LIN {X 0,Y 488.719,Z 166.606,A -85,B 0,C 180,E1 -6637.153,E2 -6637.153} C_VEL
LIN {X 0,Y 488.723,Z 166.608,A -85,B 0,C 180,E1 -6639.81,E2 -6639.81} C_VEL
LIN {X 0,Y 488.727,Z 166.608,A -85,B 0,C 180,E1 -6642.423,E2 -6642.423} C_VEL
LIN {X 0,Y 488.76,Z 166.604,A -85,B 0,C 180,E1 -6645,E2 -6645} C_VEL
LIN {X 0,Y 488.802,Z 166.598,A -85,B 0,C 180,E1 -6648.387,E2 -6648.387} C_VEL
LIN {X 0,Y 488.758,Z 166.603,A -85,B 0,C 180,E1 -6651.733,E2 -6651.733} C_VEL
LIN {X 0,Y 488.825,Z 166.593,A -85,B 0,C 180,E1 -6654.224,E2 -6654.224} C_VEL
LIN {X 0,Y 488.957,Z 166.578,A -85,B 0,C 180,E1 -6657.529,E2 -6657.529} C_VEL
LIN {X 0,Y 488.953,Z 166.579,A -85,B 0,C 180,E1 -6660.824,E2 -6660.824} C_VEL
LIN {X 0,Y 488.957,Z 166.578,A -85,B 0,C 180,E1 -6662.471,E2 -6662.471} C_VEL
LIN {X 0,Y 488.824,Z 166.594,A -85,B 0,C 180,E1 -6665.776,E2 -6665.776} C_VEL
LIN {X 0,Y 488.758,Z 166.604,A -85,B 0,C 180,E1 -6668.267,E2 -6668.267} C_VEL
LIN {X 0,Y 488.803,Z 166.597,A -85,B 0,C 180,E1 -6671.613,E2 -6671.613} C_VEL
LIN {X 0,Y 488.76,Z 166.604,A -85,B 0,C 180,E1 -6675.001,E2 -6675.001} C_VEL
LIN {X 0,Y 488.753,Z 166.606,A -85,B 0,C 180,E1 -6678.442,E2 -6678.442} C_VEL
LIN {X 0,Y 488.705,Z 166.61,A -85,B 0,C 180,E1 -6681.071,E2 -6681.071} C_VEL
LIN {X 0,Y 488.677,Z 166.615,A -85,B 0,C 180,E1 -6683.746,E2 -6683.746} C_VEL
LIN {X 0,Y 488.791,Z 166.598,A -85,B 0,C 180,E1 -6686.944,E2 -6686.944} C_VEL
LIN {X 0,Y 488.708,Z 166.61,A -85,B 0,C 180,E1 -6690.363,E2 -6690.363} C_VEL
LIN {X 0,Y 488.733,Z 166.606,A -85,B 0,C 180,E1 -6693.484,E2 -6693.484} C_VEL
LIN {X 0,Y 488.654,Z 166.616,A -85,B 0,C 180,E1 -6696.35,E2 -6696.35} C_VEL
LIN {X 0,Y 488.693,Z 166.614,A -85,B 0,C 180,E1 -6699.255,E2 -6699.255} C_VEL
LIN {X 0,Y 488.706,Z 166.608,A -85,B 0,C 180,E1 -6701.6,E2 -6701.6} C_VEL
LIN {X 0,Y 488.712,Z 166.611,A -85,B 0,C 180,E1 -6704.802,E2 -6704.802} C_VEL
LIN {X 0,Y 488.692,Z 166.612,A -85,B 0,C 180,E1 -6707.475,E2 -6707.475} C_VEL
LIN {X 0,Y 488.733,Z 166.607,A -85,B 0,C 180,E1 -6709.677,E2 -6709.677} C_VEL
LIN {X 0,Y 488.66,Z 166.618,A -85,B 0,C 180,E1 -6712.84,E2 -6712.84} C_VEL
LIN {X 0,Y 488.621,Z 166.621,A -85,B 0,C 180,E1 -6713.863,E2 -6713.863} C_VEL
LIN {X 0,Y 488.566,Z 167.341,A -85,B 0,C 180,E1 -6715.079,E2 -6715.079} C_VEL
LIN {X 0,Y 488.541,Z 171.624,A -85,B 0,C 180,E1 -6718.077,E2 -6718.077} C_VEL
LIN {X 0,Y 488.466,Z 175.456,A -85,B 0,C 180,E1 -6720.713,E2 -6720.713} C_VEL
LIN {X 0,Y 488.362,Z 179.614,A -85,B 0,C 180,E1 -6723.505,E2 -6723.505} C_VEL
LIN {X 0,Y 488.318,Z 180.585,A -85,B 0,C 180,E1 -6724.154,E2 -6724.154} C_VEL
LIN {X 0,Y 487.645,Z 181.674,A -85,B 0,C 180,E1 -6724.83,E2 -6724.83} C_VEL
LIN {X 0,Y 484.77,Z 183.623,A -85,B 0,C 180,E1 -6725.923,E2 -6725.923} C_VEL
LIN {X 0,Y 482.327,Z 185.202,A -85,B 0,C 180,E1 -6726.804,E2 -6726.804} C_VEL
LIN {X 0,Y 481.259,Z 186.339,A -85,B 0,C 180,E1 -6727.486,E2 -6727.486} C_VEL
LIN {X 0,Y 481.163,Z 186.7,A -85,B 0,C 180,E1 -6727.718,E2 -6727.718} C_VEL
LIN {X 0,Y 481.076,Z 190.806,A -85,B 0,C 180,E1 -6730.367,E2 -6730.367} C_VEL
LIN {X 0,Y 480.989,Z 195.029,A -85,B 0,C 180,E1 -6733.009,E2 -6733.009} C_VEL
LIN {X 0,Y 480.962,Z 198.538,A -85,B 0,C 180,E1 -6735.13,E2 -6735.13} C_VEL
LIN {X 0,Y 483.732,Z 212.205,A -85,B 0,C 180,E1 -6735.607,E2 -6735.607} C_VEL
LIN {X 0,Y 484.026,Z 214.848,A -85,B 0,C 180,E1 -6735.71,E2 -6735.71} C_VEL
LIN {X 0,Y 483.673,Z 226.76,A -85,B 0,C 180,E1 -6736.235,E2 -6736.235} C_VEL
LIN {X 0,Y 483.3,Z 238.299,A -85,B 0,C 180,E1 -6736.914,E2 -6736.914} C_VEL
LIN {X 0,Y 482.921,Z 248.978,A -85,B 0,C 180,E1 -6737.711,E2 -6737.711} C_VEL
LIN {X 0,Y 482.468,Z 259.22,A -85,B 0,C 180,E1 -6738.659,E2 -6738.659} C_VEL
LIN {X 0,Y 482.079,Z 268.408,A -85,B 0,C 180,E1 -6739.713,E2 -6739.713} C_VEL
LIN {X 0,Y 481.679,Z 277.326,A -85,B 0,C 180,E1 -6740.976,E2 -6740.976} C_VEL
LIN {X 0,Y 481.347,Z 284.505,A -85,B 0,C 180,E1 -6742.238,E2 -6742.238} C_VEL
LIN {X 0,Y 481.17,Z 290.612,A -85,B 0,C 180,E1 -6743.598,E2 -6743.598} C_VEL
LIN {X 0,Y 480.918,Z 295.37,A -85,B 0,C 180,E1 -6744.97,E2 -6744.97} C_VEL
LIN {X 0,Y 480.976,Z 297.654,A -85,B 0,C 180,E1 -6745.81,E2 -6745.81} C_VEL
LIN {X 0,Y 480.936,Z 299.516,A -85,B 0,C 180,E1 -6746.649,E2 -6746.649} C_VEL
LIN {X 0,Y 480.855,Z 300.922,A -85,B 0,C 180,E1 -6747.487,E2 -6747.487} C_VEL
LIN {X 0,Y 480.824,Z 301.92,A -85,B 0,C 180,E1 -6748.325,E2 -6748.325} C_VEL
LIN {X 0,Y 480.746,Z 302.773,A -85,B 0,C 180,E1 -6750,E2 -6750} C_VEL
LIN {X 0,Y 480.761,Z 302.588,A -85,B 0,C 180,E1 -6750.838,E2 -6750.838} C_VEL
LIN {X 0,Y 480.825,Z 302.004,A -85,B 0,C 180,E1 -6751.675,E2 -6751.675} C_VEL
LIN {X 0,Y 480.936,Z 299.683,A -85,B 0,C 180,E1 -6753.351,E2 -6753.351} C_VEL
LIN {X 0,Y 480.925,Z 296.824,A -85,B 0,C 180,E1 -6754.61,E2 -6754.61} C_VEL
LIN {X 0,Y 481.147,Z 292.94,A -85,B 0,C 180,E1 -6755.869,E2 -6755.869} C_VEL
LIN {X 0,Y 481.199,Z 287.935,A -85,B 0,C 180,E1 -6757.132,E2 -6757.132} C_VEL
LIN {X 0,Y 481.492,Z 281.631,A -85,B 0,C 180,E1 -6758.393,E2 -6758.393} C_VEL
LIN {X 0,Y 481.822,Z 273.737,A -85,B 0,C 180,E1 -6759.657,E2 -6759.657} C_VEL
LIN {X 0,Y 482.161,Z 265.691,A -85,B 0,C 180,E1 -6760.711,E2 -6760.711} C_VEL
LIN {X 0,Y 482.609,Z 255.869,A -85,B 0,C 180,E1 -6761.764,E2 -6761.764} C_VEL
LIN {X 0,Y 483,Z 246.206,A -85,B 0,C 180,E1 -6762.607,E2 -6762.607} C_VEL
LIN {X 0,Y 483.345,Z 235.574,A -85,B 0,C 180,E1 -6763.357,E2 -6763.357} C_VEL
LIN {X 0,Y 483.791,Z 223.171,A -85,B 0,C 180,E1 -6764.029,E2 -6764.029} C_VEL
LIN {X 0,Y 483.955,Z 213.248,A -85,B 0,C 180,E1 -6764.44,E2 -6764.44} C_VEL
LIN {X 0,Y 481.334,Z 200.392,A -85,B 0,C 180,E1 -6764.902,E2 -6764.902} C_VEL
LIN {X 0,Y 480.987,Z 198.508,A -85,B 0,C 180,E1 -6764.978,E2 -6764.978} C_VEL
LIN {X 0,Y 481.039,Z 193.157,A -85,B 0,C 180,E1 -6768.258,E2 -6768.258} C_VEL
LIN {X 0,Y 481.141,Z 188.161,A -85,B 0,C 180,E1 -6771.418,E2 -6771.418} C_VEL
LIN {X 0,Y 481.274,Z 184.043,A -85,B 0,C 180,E1 -6774.135,E2 -6774.135} C_VEL
LIN {X 0,Y 481.315,Z 179.709,A -85,B 0,C 180,E1 -6777.038,E2 -6777.038} C_VEL
LIN {X 0,Y 481.425,Z 175.715,A -85,B 0,C 180,E1 -6779.758,E2 -6779.758} C_VEL
LIN {X 0,Y 481.504,Z 171.509,A -85,B 0,C 180,E1 -6782.687,E2 -6782.687} C_VEL
LIN {X 0,Y 481.566,Z 168.004,A -85,B 0,C 180,E1 -6785.187,E2 -6785.187} C_VEL
LIN {X 0,Y 481.547,Z 167.504,A -85,B 0,C 180,E1 -6785.717,E2 -6785.717} C_VEL
LIN {X 0,Y 481.629,Z 167.493,A -85,B 0,C 180,E1 -6788.863,E2 -6788.863} C_VEL
LIN {X 0,Y 481.637,Z 167.492,A -85,B 0,C 180,E1 -6791.91,E2 -6791.91} C_VEL
LIN {X 0,Y 481.656,Z 167.488,A -85,B 0,C 180,E1 -6794.458,E2 -6794.458} C_VEL
LIN {X 0,Y 481.649,Z 167.487,A -85,B 0,C 180,E1 -6797.839,E2 -6797.839} C_VEL
LIN {X 0,Y 481.657,Z 167.49,A -85,B 0,C 180,E1 -6800.655,E2 -6800.655} C_VEL
LIN {X 0,Y 481.611,Z 167.493,A -85,B 0,C 180,E1 -6803.379,E2 -6803.379} C_VEL
LIN {X 0,Y 481.671,Z 167.487,A -85,B 0,C 180,E1 -6806.327,E2 -6806.327} C_VEL
LIN {X 0,Y 481.652,Z 167.489,A -85,B 0,C 180,E1 -6809.417,E2 -6809.417} C_VEL
LIN {X 0,Y 481.701,Z 167.482,A -85,B 0,C 180,E1 -6812.168,E2 -6812.168} C_VEL
LIN {X 0,Y 481.694,Z 167.48,A -85,B 0,C 180,E1 -6814.968,E2 -6814.968} C_VEL
LIN {X 0,Y 481.649,Z 167.49,A -85,B 0,C 180,E1 -6817.705,E2 -6817.705} C_VEL
LIN {X 0,Y 481.705,Z 167.481,A -85,B 0,C 180,E1 -6820.393,E2 -6820.393} C_VEL
LIN {X 0,Y 481.681,Z 167.485,A -85,B 0,C 180,E1 -6823.033,E2 -6823.033} C_VEL
LIN {X 0,Y 481.691,Z 167.483,A -85,B 0,C 180,E1 -6825.639,E2 -6825.639} C_VEL
LIN {X 0,Y 481.752,Z 167.477,A -85,B 0,C 180,E1 -6828.215,E2 -6828.215} C_VEL
LIN {X 0,Y 481.721,Z 167.482,A -85,B 0,C 180,E1 -6831.611,E2 -6831.611} C_VEL
LIN {X 0,Y 481.784,Z 167.471,A -85,B 0,C 180,E1 -6834.139,E2 -6834.139} C_VEL
LIN {X 0,Y 481.925,Z 167.454,A -85,B 0,C 180,E1 -6837.492,E2 -6837.492} C_VEL
LIN {X 0,Y 481.907,Z 167.456,A -85,B 0,C 180,E1 -6840.836,E2 -6840.836} C_VEL
LIN {X 0,Y 481.927,Z 167.453,A -85,B 0,C 180,E1 -6842.507,E2 -6842.507} C_VEL
LIN {X 0,Y 481.787,Z 167.469,A -85,B 0,C 180,E1 -6845.861,E2 -6845.861} C_VEL
LIN {X 0,Y 481.72,Z 167.48,A -85,B 0,C 180,E1 -6848.389,E2 -6848.389} C_VEL
LIN {X 0,Y 481.795,Z 167.47,A -85,B 0,C 180,E1 -6851.784,E2 -6851.784} C_VEL
LIN {X 0,Y 481.744,Z 167.478,A -85,B 0,C 180,E1 -6855.224,E2 -6855.224} C_VEL
LIN {X 0,Y 481.709,Z 167.484,A -85,B 0,C 180,E1 -6858.722,E2 -6858.722} C_VEL
LIN {X 0,Y 481.646,Z 167.487,A -85,B 0,C 180,E1 -6861.395,E2 -6861.395} C_VEL
LIN {X 0,Y 481.658,Z 167.491,A -85,B 0,C 180,E1 -6864.114,E2 -6864.114} C_VEL
LIN {X 0,Y 481.747,Z 167.476,A -85,B 0,C 180,E1 -6867.139,E2 -6867.139} C_VEL
LIN {X 0,Y 481.68,Z 167.485,A -85,B 0,C 180,E1 -6869.741,E2 -6869.741} C_VEL
LIN {X 0,Y 481.673,Z 167.486,A -85,B 0,C 180,E1 -6872.674,E2 -6872.674} C_VEL
LIN {X 0,Y 481.621,Z 167.494,A -85,B 0,C 180,E1 -6875.711,E2 -6875.711} C_VEL
LIN {X 0,Y 481.632,Z 167.488,A -85,B 0,C 180,E1 -6878.863,E2 -6878.863} C_VEL
LIN {X 0,Y 481.654,Z 167.487,A -85,B 0,C 180,E1 -6881.913,E2 -6881.913} C_VEL
LIN {X 0,Y 481.656,Z 167.491,A -85,B 0,C 180,E1 -6884.458,E2 -6884.458} C_VEL
LIN {X 0,Y 481.649,Z 167.489,A -85,B 0,C 180,E1 -6887.839,E2 -6887.839} C_VEL
LIN {X 0,Y 481.694,Z 167.487,A -85,B 0,C 180,E1 -6891.143,E2 -6891.143} C_VEL
LIN {X 0,Y 482.385,Z 171.769,A -85,B 0,C 180,E1 -6893.32,E2 -6893.32} C_VEL
LIN {X 0,Y 482.593,Z 176.26,A -85,B 0,C 180,E1 -6895.392,E2 -6895.392} C_VEL
LIN {X 0,Y 482.336,Z 183.028,A -85,B 0,C 180,E1 -6898.362,E2 -6898.362} C_VEL
LIN {X 0,Y 482.081,Z 189.813,A -85,B 0,C 180,E1 -6901.243,E2 -6901.243} C_VEL
LIN {X 0,Y 481.84,Z 196.575,A -85,B 0,C 180,E1 -6904.051,E2 -6904.051} C_VEL
LIN {X 0,Y 481.638,Z 204.537,A -85,B 0,C 180,E1 -6907.257,E2 -6907.257} C_VEL
LIN {X 0,Y 481.474,Z 212.483,A -85,B 0,C 180,E1 -6910.383,E2 -6910.383} C_VEL
LIN {X 0,Y 481.232,Z 221.5,A -85,B 0,C 180,E1 -6913.89,E2 -6913.89} C_VEL
LIN {X 0,Y 481.158,Z 224.491,A -85,B 0,C 180,E1 -6915.055,E2 -6915.055} C_VEL
LIN {X 0,Y 483.558,Z 238.307,A -85,B 0,C 180,E1 -6915.494,E2 -6915.494} C_VEL
LIN {X 0,Y 483.944,Z 242.497,A -85,B 0,C 180,E1 -6915.653,E2 -6915.653} C_VEL
LIN {X 0,Y 483.598,Z 254.507,A -85,B 0,C 180,E1 -6916.179,E2 -6916.179} C_VEL
LIN {X 0,Y 483.096,Z 266.675,A -85,B 0,C 180,E1 -6916.893,E2 -6916.893} C_VEL
LIN {X 0,Y 482.718,Z 277.483,A -85,B 0,C 180,E1 -6917.706,E2 -6917.706} C_VEL
LIN {X 0,Y 482.312,Z 287.644,A -85,B 0,C 180,E1 -6918.655,E2 -6918.655} C_VEL
LIN {X 0,Y 481.875,Z 296.784,A -85,B 0,C 180,E1 -6919.708,E2 -6919.708} C_VEL
LIN {X 0,Y 481.531,Z 305.687,A -85,B 0,C 180,E1 -6920.973,E2 -6920.973} C_VEL
LIN {X 0,Y 481.208,Z 312.848,A -85,B 0,C 180,E1 -6922.236,E2 -6922.236} C_VEL
LIN {X 0,Y 481.048,Z 318.356,A -85,B 0,C 180,E1 -6923.447,E2 -6923.447} C_VEL
LIN {X 0,Y 480.998,Z 322.372,A -85,B 0,C 180,E1 -6924.55,E2 -6924.55} C_VEL
LIN {X 0,Y 480.847,Z 325.957,A -85,B 0,C 180,E1 -6925.809,E2 -6925.809} C_VEL
LIN {X 0,Y 480.891,Z 327.806,A -85,B 0,C 180,E1 -6926.648,E2 -6926.648} C_VEL
LIN {X 0,Y 480.79,Z 330.182,A -85,B 0,C 180,E1 -6928.325,E2 -6928.325} C_VEL
LIN {X 0,Y 480.743,Z 331,A -85,B 0,C 180,E1 -6930,E2 -6930} C_VEL
LIN {X 0,Y 480.79,Z 330.184,A -85,B 0,C 180,E1 -6931.675,E2 -6931.675} C_VEL
LIN {X 0,Y 480.891,Z 327.81,A -85,B 0,C 180,E1 -6933.351,E2 -6933.351} C_VEL
LIN {X 0,Y 480.854,Z 324.896,A -85,B 0,C 180,E1 -6934.611,E2 -6934.611} C_VEL
LIN {X 0,Y 481.023,Z 320.949,A -85,B 0,C 180,E1 -6935.87,E2 -6935.87} C_VEL
LIN {X 0,Y 481.116,Z 314.877,A -85,B 0,C 180,E1 -6937.343,E2 -6937.343} C_VEL
LIN {X 0,Y 481.426,Z 308.237,A -85,B 0,C 180,E1 -6938.605,E2 -6938.605} C_VEL
LIN {X 0,Y 481.755,Z 299.994,A -85,B 0,C 180,E1 -6939.87,E2 -6939.87} C_VEL
LIN {X 0,Y 482.074,Z 291.542,A -85,B 0,C 180,E1 -6940.925,E2 -6940.925} C_VEL
LIN {X 0,Y 482.564,Z 281.094,A -85,B 0,C 180,E1 -6941.978,E2 -6941.978} C_VEL
LIN {X 0,Y 482.966,Z 269.881,A -85,B 0,C 180,E1 -6942.887,E2 -6942.887} C_VEL
LIN {X 0,Y 483.353,Z 259.409,A -85,B 0,C 180,E1 -6943.559,E2 -6943.559} C_VEL
LIN {X 0,Y 483.807,Z 247.77,A -85,B 0,C 180,E1 -6944.136,E2 -6944.136} C_VEL
LIN {X 0,Y 483.769,Z 239.834,A -85,B 0,C 180,E1 -6944.446,E2 -6944.446} C_VEL
LIN {X 0,Y 481.599,Z 226.955,A -85,B 0,C 180,E1 -6944.877,E2 -6944.877} C_VEL
LIN {X 0,Y 481.163,Z 224.423,A -85,B 0,C 180,E1 -6944.972,E2 -6944.972} C_VEL
LIN {X 0,Y 481.347,Z 215.691,A -85,B 0,C 180,E1 -6948.369,E2 -6948.369} C_VEL
LIN {X 0,Y 481.52,Z 209.151,A -85,B 0,C 180,E1 -6950.915,E2 -6950.915} C_VEL
LIN {X 0,Y 481.715,Z 201.065,A -85,B 0,C 180,E1 -6954.111,E2 -6954.111} C_VEL
LIN {X 0,Y 481.954,Z 193.576,A -85,B 0,C 180,E1 -6957.186,E2 -6957.186} C_VEL
LIN {X 0,Y 482.23,Z 186.418,A -85,B 0,C 180,E1 -6960.185,E2 -6960.185} C_VEL
LIN {X 0,Y 482.447,Z 179.637,A -85,B 0,C 180,E1 -6963.112,E2 -6963.112} C_VEL
LIN {X 0,Y 482.598,Z 174.007,A -85,B 0,C 180,E1 -6965.627,E2 -6965.627} C_VEL
LIN {X 0,Y 481.943,Z 168.93,A -85,B 0,C 180,E1 -6968.051,E2 -6968.051} C_VEL
LIN {X 0,Y 481.692,Z 167.488,A -85,B 0,C 180,E1 -6968.857,E2 -6968.857} C_VEL
LIN {X 0,Y 481.647,Z 167.492,A -85,B 0,C 180,E1 -6972.16,E2 -6972.16} C_VEL
LIN {X 0,Y 481.653,Z 167.489,A -85,B 0,C 180,E1 -6975.542,E2 -6975.542} C_VEL
LIN {X 0,Y 481.655,Z 167.489,A -85,B 0,C 180,E1 -6978.958,E2 -6978.958} C_VEL
LIN {X 0,Y 481.63,Z 167.491,A -85,B 0,C 180,E1 -6981.996,E2 -6981.996} C_VEL
LIN {X 0,Y 481.683,Z 167.484,A -85,B 0,C 180,E1 -6985.317,E2 -6985.317} C_VEL
LIN {X 0,Y 481.643,Z 167.489,A -85,B 0,C 180,E1 -6988.311,E2 -6988.311} C_VEL
LIN {X 0,Y 481.699,Z 167.483,A -85,B 0,C 180,E1 -6991.218,E2 -6991.218} C_VEL
LIN {X 0,Y 481.687,Z 167.486,A -85,B 0,C 180,E1 -6994.042,E2 -6994.042} C_VEL
LIN {X 0,Y 481.672,Z 167.483,A -85,B 0,C 180,E1 -6996.812,E2 -6996.812} C_VEL
LIN {X 0,Y 481.693,Z 167.487,A -85,B 0,C 180,E1 -6999.503,E2 -6999.503} C_VEL
LIN {X 0,Y 481.702,Z 167.482,A -85,B 0,C 180,E1 -7002.158,E2 -7002.158} C_VEL
LIN {X 0,Y 481.741,Z 167.479,A -85,B 0,C 180,E1 -7004.776,E2 -7004.776} C_VEL
LIN {X 0,Y 481.748,Z 167.476,A -85,B 0,C 180,E1 -7008.215,E2 -7008.215} C_VEL
LIN {X 0,Y 481.717,Z 167.481,A -85,B 0,C 180,E1 -7011.611,E2 -7011.611} C_VEL
LIN {X 0,Y 481.784,Z 167.469,A -85,B 0,C 180,E1 -7014.139,E2 -7014.139} C_VEL
LIN {X 0,Y 481.924,Z 167.454,A -85,B 0,C 180,E1 -7017.493,E2 -7017.493} C_VEL
LIN {X 0,Y 481.904,Z 167.457,A -85,B 0,C 180,E1 -7020.836,E2 -7020.836} C_VEL
LIN {X 0,Y 481.924,Z 167.454,A -85,B 0,C 180,E1 -7022.508,E2 -7022.508} C_VEL
LIN {X 0,Y 481.783,Z 167.471,A -85,B 0,C 180,E1 -7025.861,E2 -7025.861} C_VEL
LIN {X 0,Y 481.718,Z 167.482,A -85,B 0,C 180,E1 -7028.389,E2 -7028.389} C_VEL
LIN {X 0,Y 481.748,Z 167.476,A -85,B 0,C 180,E1 -7031.785,E2 -7031.785} C_VEL
LIN {X 0,Y 481.741,Z 167.478,A -85,B 0,C 180,E1 -7035.224,E2 -7035.224} C_VEL
LIN {X 0,Y 481.71,Z 167.482,A -85,B 0,C 180,E1 -7038.722,E2 -7038.722} C_VEL
LIN {X 0,Y 481.643,Z 167.488,A -85,B 0,C 180,E1 -7041.395,E2 -7041.395} C_VEL
LIN {X 0,Y 481.659,Z 167.489,A -85,B 0,C 180,E1 -7044.114,E2 -7044.114} C_VEL
LIN {X 0,Y 481.745,Z 167.476,A -85,B 0,C 180,E1 -7047.14,E2 -7047.14} C_VEL
LIN {X 0,Y 481.677,Z 167.485,A -85,B 0,C 180,E1 -7049.741,E2 -7049.741} C_VEL
LIN {X 0,Y 481.67,Z 167.487,A -85,B 0,C 180,E1 -7052.675,E2 -7052.675} C_VEL
LIN {X 0,Y 481.62,Z 167.495,A -85,B 0,C 180,E1 -7055.711,E2 -7055.711} C_VEL
LIN {X 0,Y 481.634,Z 167.49,A -85,B 0,C 180,E1 -7058.863,E2 -7058.863} C_VEL
LIN {X 0,Y 481.652,Z 167.486,A -85,B 0,C 180,E1 -7061.913,E2 -7061.913} C_VEL
LIN {X 0,Y 481.659,Z 167.488,A -85,B 0,C 180,E1 -7064.458,E2 -7064.458} C_VEL
LIN {X 0,Y 481.647,Z 167.489,A -85,B 0,C 180,E1 -7067.84,E2 -7067.84} C_VEL
LIN {X 0,Y 481.656,Z 167.488,A -85,B 0,C 180,E1 -7070.655,E2 -7070.655} C_VEL
LIN {X 0,Y 481.602,Z 167.498,A -85,B 0,C 180,E1 -7073.381,E2 -7073.381} C_VEL
LIN {X 0,Y 481.515,Z 167.507,A -85,B 0,C 180,E1 -7074.28,E2 -7074.28} C_VEL
LIN {X 0,Y 481.515,Z 168.566,A -85,B 0,C 180,E1 -7075.304,E2 -7075.304} C_VEL
LIN {X 0,Y 481.468,Z 172.792,A -85,B 0,C 180,E1 -7078.299,E2 -7078.299} C_VEL
LIN {X 0,Y 481.409,Z 176.97,A -85,B 0,C 180,E1 -7081.2,E2 -7081.2} C_VEL
LIN {X 0,Y 481.268,Z 181.295,A -85,B 0,C 180,E1 -7084.134,E2 -7084.134} C_VEL
LIN {X 0,Y 481.228,Z 185.508,A -85,B 0,C 180,E1 -7086.937,E2 -7086.937} C_VEL
LIN {X 0,Y 481.163,Z 186.7,A -85,B 0,C 180,E1 -7087.718,E2 -7087.718} C_VEL
LIN {X 0,Y 480.459,Z 187.815,A -85,B 0,C 180,E1 -7088.404,E2 -7088.404} C_VEL
LIN {X 0,Y 477.551,Z 189.802,A -85,B 0,C 180,E1 -7089.513,E2 -7089.513} C_VEL
LIN {X 0,Y 475.106,Z 191.418,A -85,B 0,C 180,E1 -7090.407,E2 -7090.407} C_VEL
LIN {X 0,Y 474.057,Z 192.597,A -85,B 0,C 180,E1 -7091.099,E2 -7091.099} C_VEL
LIN {X 0,Y 473.972,Z 192.975,A -85,B 0,C 180,E1 -7091.334,E2 -7091.334} C_VEL
LIN {X 0,Y 473.925,Z 198.725,A -85,B 0,C 180,E1 -7094.9,E2 -7094.9} C_VEL
LIN {X 0,Y 476.875,Z 213.241,A -85,B 0,C 180,E1 -7095.425,E2 -7095.425} C_VEL
LIN {X 0,Y 477.075,Z 217.711,A -85,B 0,C 180,E1 -7095.606,E2 -7095.606} C_VEL
LIN {X 0,Y 476.726,Z 228.965,A -85,B 0,C 180,E1 -7096.14,E2 -7096.14} C_VEL
LIN {X 0,Y 476.267,Z 240.238,A -85,B 0,C 180,E1 -7096.835,E2 -7096.835} C_VEL
LIN {X 0,Y 475.87,Z 251.672,A -85,B 0,C 180,E1 -7097.743,E2 -7097.743} C_VEL
LIN {X 0,Y 475.424,Z 261.398,A -85,B 0,C 180,E1 -7098.705,E2 -7098.705} C_VEL
LIN {X 0,Y 474.994,Z 270.245,A -85,B 0,C 180,E1 -7099.773,E2 -7099.773} C_VEL
LIN {X 0,Y 474.595,Z 278.875,A -85,B 0,C 180,E1 -7101.055,E2 -7101.055} C_VEL
LIN {X 0,Y 474.257,Z 285.754,A -85,B 0,C 180,E1 -7102.336,E2 -7102.336} C_VEL
LIN {X 0,Y 474.105,Z 291.155,A -85,B 0,C 180,E1 -7103.59,E2 -7103.59} C_VEL
LIN {X 0,Y 473.858,Z 295.585,A -85,B 0,C 180,E1 -7104.895,E2 -7104.895} C_VEL
LIN {X 0,Y 473.88,Z 297.869,A -85,B 0,C 180,E1 -7105.748,E2 -7105.748} C_VEL
LIN {X 0,Y 473.865,Z 299.73,A -85,B 0,C 180,E1 -7106.599,E2 -7106.599} C_VEL
LIN {X 0,Y 473.773,Z 301.136,A -85,B 0,C 180,E1 -7107.45,E2 -7107.45} C_VEL
LIN {X 0,Y 473.69,Z 302.75,A -85,B 0,C 180,E1 -7109.15,E2 -7109.15} C_VEL
LIN {X 0,Y 473.672,Z 302.986,A -85,B 0,C 180,E1 -7110,E2 -7110} C_VEL
LIN {X 0,Y 473.69,Z 302.8,A -85,B 0,C 180,E1 -7110.85,E2 -7110.85} C_VEL
LIN {X 0,Y 473.773,Z 301.251,A -85,B 0,C 180,E1 -7112.551,E2 -7112.551} C_VEL
LIN {X 0,Y 473.865,Z 299.895,A -85,B 0,C 180,E1 -7113.401,E2 -7113.401} C_VEL
LIN {X 0,Y 473.834,Z 297.036,A -85,B 0,C 180,E1 -7114.679,E2 -7114.679} C_VEL
LIN {X 0,Y 474.092,Z 293.151,A -85,B 0,C 180,E1 -7115.956,E2 -7115.956} C_VEL
LIN {X 0,Y 474.149,Z 288.146,A -85,B 0,C 180,E1 -7117.238,E2 -7117.238} C_VEL
LIN {X 0,Y 474.445,Z 281.842,A -85,B 0,C 180,E1 -7118.519,E2 -7118.519} C_VEL
LIN {X 0,Y 474.827,Z 273.947,A -85,B 0,C 180,E1 -7119.8,E2 -7119.8} C_VEL
LIN {X 0,Y 475.179,Z 265.9,A -85,B 0,C 180,E1 -7120.87,E2 -7120.87} C_VEL
LIN {X 0,Y 475.668,Z 256.077,A -85,B 0,C 180,E1 -7121.938,E2 -7121.938} C_VEL
LIN {X 0,Y 476.073,Z 246.414,A -85,B 0,C 180,E1 -7122.794,E2 -7122.794} C_VEL
LIN {X 0,Y 476.442,Z 235.888,A -85,B 0,C 180,E1 -7123.548,E2 -7123.548} C_VEL
LIN {X 0,Y 476.929,Z 223.373,A -85,B 0,C 180,E1 -7124.236,E2 -7124.236} C_VEL
LIN {X 0,Y 477.077,Z 214.3,A -85,B 0,C 180,E1 -7124.623,E2 -7124.623} C_VEL
LIN {X 0,Y 474.36,Z 200.975,A -85,B 0,C 180,E1 -7125.117,E2 -7125.117} C_VEL
LIN {X 0,Y 473.934,Z 198.727,A -85,B 0,C 180,E1 -7125.19,E2 -7125.19} C_VEL
LIN {X 0,Y 473.973,Z 193.584,A -85,B 0,C 180,E1 -7128.38,E2 -7128.38} C_VEL
LIN {X 0,Y 474.085,Z 188.324,A -85,B 0,C 180,E1 -7131.753,E2 -7131.753} C_VEL
LIN {X 0,Y 474.199,Z 184.193,A -85,B 0,C 180,E1 -7134.518,E2 -7134.518} C_VEL
LIN {X 0,Y 474.278,Z 180.026,A -85,B 0,C 180,E1 -7137.346,E2 -7137.346} C_VEL
LIN {X 0,Y 474.381,Z 175.832,A -85,B 0,C 180,E1 -7140.246,E2 -7140.246} C_VEL
LIN {X 0,Y 474.463,Z 171.613,A -85,B 0,C 180,E1 -7143.234,E2 -7143.234} C_VEL
LIN {X 0,Y 474.505,Z 168.562,A -85,B 0,C 180,E1 -7145.45,E2 -7145.45} C_VEL
LIN {X 0,Y 474.59,Z 168.368,A -85,B 0,C 180,E1 -7148.292,E2 -7148.292} C_VEL
LIN {X 0,Y 474.607,Z 168.367,A -85,B 0,C 180,E1 -7150.956,E2 -7150.956} C_VEL
LIN {X 0,Y 474.604,Z 168.366,A -85,B 0,C 180,E1 -7154.106,E2 -7154.106} C_VEL
LIN {X 0,Y 474.616,Z 168.367,A -85,B 0,C 180,E1 -7157.066,E2 -7157.066} C_VEL
LIN {X 0,Y 474.619,Z 168.364,A -85,B 0,C 180,E1 -7159.342,E2 -7159.342} C_VEL
LIN {X 0,Y 474.593,Z 168.366,A -85,B 0,C 180,E1 -7161.707,E2 -7161.707} C_VEL
LIN {X 0,Y 474.614,Z 168.365,A -85,B 0,C 180,E1 -7164.725,E2 -7164.725} C_VEL
LIN {X 0,Y 474.636,Z 168.363,A -85,B 0,C 180,E1 -7167.788,E2 -7167.788} C_VEL
LIN {X 0,Y 474.625,Z 168.365,A -85,B 0,C 180,E1 -7170.884,E2 -7170.884} C_VEL
LIN {X 0,Y 474.655,Z 168.358,A -85,B 0,C 180,E1 -7173.628,E2 -7173.628} C_VEL
LIN {X 0,Y 474.636,Z 168.361,A -85,B 0,C 180,E1 -7176.642,E2 -7176.642} C_VEL
LIN {X 0,Y 474.655,Z 168.36,A -85,B 0,C 180,E1 -7180.089,E2 -7180.089} C_VEL
LIN {X 0,Y 474.64,Z 168.362,A -85,B 0,C 180,E1 -7182.774,E2 -7182.774} C_VEL
LIN {X 0,Y 474.649,Z 168.361,A -85,B 0,C 180,E1 -7185.421,E2 -7185.421} C_VEL
LIN {X 0,Y 474.705,Z 168.356,A -85,B 0,C 180,E1 -7188.038,E2 -7188.038} C_VEL
LIN {X 0,Y 474.696,Z 168.358,A -85,B 0,C 180,E1 -7191.486,E2 -7191.486} C_VEL
LIN {X 0,Y 474.745,Z 168.347,A -85,B 0,C 180,E1 -7194.052,E2 -7194.052} C_VEL
LIN {X 0,Y 474.891,Z 168.33,A -85,B 0,C 180,E1 -7197.455,E2 -7197.455} C_VEL
LIN {X 0,Y 474.913,Z 168.328,A -85,B 0,C 180,E1 -7200,E2 -7200} C_VEL
LIN {X 0,Y 474.893,Z 168.33,A -85,B 0,C 180,E1 -7202.545,E2 -7202.545} C_VEL
LIN {X 0,Y 474.748,Z 168.346,A -85,B 0,C 180,E1 -7205.948,E2 -7205.948} C_VEL
LIN {X 0,Y 474.695,Z 168.356,A -85,B 0,C 180,E1 -7208.514,E2 -7208.514} C_VEL
LIN {X 0,Y 474.739,Z 168.35,A -85,B 0,C 180,E1 -7211.962,E2 -7211.962} C_VEL
LIN {X 0,Y 474.681,Z 168.357,A -85,B 0,C 180,E1 -7215.768,E2 -7215.768} C_VEL
LIN {X 0,Y 474.664,Z 168.359,A -85,B 0,C 180,E1 -7219.01,E2 -7219.01} C_VEL
LIN {X 0,Y 474.589,Z 168.367,A -85,B 0,C 180,E1 -7221.729,E2 -7221.729} C_VEL
LIN {X 0,Y 474.639,Z 168.361,A -85,B 0,C 180,E1 -7224.494,E2 -7224.494} C_VEL
LIN {X 0,Y 474.682,Z 168.357,A -85,B 0,C 180,E1 -7227.334,E2 -7227.334} C_VEL
LIN {X 0,Y 474.606,Z 168.366,A -85,B 0,C 180,E1 -7230.23,E2 -7230.23} C_VEL
LIN {X 0,Y 474.635,Z 168.363,A -85,B 0,C 180,E1 -7233.221,E2 -7233.221} C_VEL
LIN {X 0,Y 474.573,Z 168.369,A -85,B 0,C 180,E1 -7236.325,E2 -7236.325} C_VEL
LIN {X 0,Y 474.612,Z 168.367,A -85,B 0,C 180,E1 -7239.645,E2 -7239.645} C_VEL
LIN {X 0,Y 474.625,Z 168.363,A -85,B 0,C 180,E1 -7242.237,E2 -7242.237} C_VEL
LIN {X 0,Y 474.618,Z 168.365,A -85,B 0,C 180,E1 -7245.298,E2 -7245.298} C_VEL
LIN {X 0,Y 474.622,Z 168.367,A -85,B 0,C 180,E1 -7248.215,E2 -7248.215} C_VEL
LIN {X 0,Y 474.669,Z 168.49,A -85,B 0,C 180,E1 -7251.073,E2 -7251.073} C_VEL
LIN {X 0,Y 475.482,Z 173.93,A -85,B 0,C 180,E1 -7253.755,E2 -7253.755} C_VEL
LIN {X 0,Y 475.547,Z 178.464,A -85,B 0,C 180,E1 -7255.854,E2 -7255.854} C_VEL
LIN {X 0,Y 475.236,Z 185.713,A -85,B 0,C 180,E1 -7259.063,E2 -7259.063} C_VEL
LIN {X 0,Y 474.996,Z 193.082,A -85,B 0,C 180,E1 -7262.22,E2 -7262.22} C_VEL
LIN {X 0,Y 474.69,Z 200.964,A -85,B 0,C 180,E1 -7265.509,E2 -7265.509} C_VEL
LIN {X 0,Y 474.5,Z 207.801,A -85,B 0,C 180,E1 -7268.267,E2 -7268.267} C_VEL
LIN {X 0,Y 474.345,Z 214.617,A -85,B 0,C 180,E1 -7270.976,E2 -7270.976} C_VEL
LIN {X 0,Y 474.166,Z 223.676,A -85,B 0,C 180,E1 -7274.526,E2 -7274.526} C_VEL
LIN {X 0,Y 474.119,Z 224.452,A -85,B 0,C 180,E1 -7274.827,E2 -7274.827} C_VEL
LIN {X 0,Y 476.543,Z 238.307,A -85,B 0,C 180,E1 -7275.275,E2 -7275.275} C_VEL
LIN {X 0,Y 477.056,Z 242.498,A -85,B 0,C 180,E1 -7275.442,E2 -7275.442} C_VEL
LIN {X 0,Y 476.706,Z 254.506,A -85,B 0,C 180,E1 -7275.975,E2 -7275.975} C_VEL
LIN {X 0,Y 476.176,Z 266.674,A -85,B 0,C 180,E1 -7276.699,E2 -7276.699} C_VEL
LIN {X 0,Y 475.753,Z 277.666,A -85,B 0,C 180,E1 -7277.538,E2 -7277.538} C_VEL
LIN {X 0,Y 475.353,Z 287.644,A -85,B 0,C 180,E1 -7278.487,E2 -7278.487} C_VEL
LIN {X 0,Y 474.877,Z 296.784,A -85,B 0,C 180,E1 -7279.555,E2 -7279.555} C_VEL
LIN {X 0,Y 474.482,Z 305.686,A -85,B 0,C 180,E1 -7280.838,E2 -7280.838} C_VEL
LIN {X 0,Y 474.153,Z 312.847,A -85,B 0,C 180,E1 -7282.119,E2 -7282.119} C_VEL
LIN {X 0,Y 473.973,Z 318.738,A -85,B 0,C 180,E1 -7283.449,E2 -7283.449} C_VEL
LIN {X 0,Y 473.846,Z 323.676,A -85,B 0,C 180,E1 -7284.894,E2 -7284.894} C_VEL
LIN {X 0,Y 473.752,Z 325.957,A -85,B 0,C 180,E1 -7285.746,E2 -7285.746} C_VEL
LIN {X 0,Y 473.799,Z 327.806,A -85,B 0,C 180,E1 -7286.598,E2 -7286.598} C_VEL
LIN {X 0,Y 473.695,Z 330.182,A -85,B 0,C 180,E1 -7288.299,E2 -7288.299} C_VEL
LIN {X 0,Y 473.688,Z 330.785,A -85,B 0,C 180,E1 -7289.15,E2 -7289.15} C_VEL
LIN {X 0,Y 473.669,Z 331,A -85,B 0,C 180,E1 -7290,E2 -7290} C_VEL
LIN {X 0,Y 473.688,Z 330.786,A -85,B 0,C 180,E1 -7290.85,E2 -7290.85} C_VEL
LIN {X 0,Y 473.724,Z 329.196,A -85,B 0,C 180,E1 -7292.551,E2 -7292.551} C_VEL
LIN {X 0,Y 473.799,Z 327.81,A -85,B 0,C 180,E1 -7293.401,E2 -7293.401} C_VEL
LIN {X 0,Y 473.776,Z 324.896,A -85,B 0,C 180,E1 -7294.68,E2 -7294.68} C_VEL
LIN {X 0,Y 473.942,Z 320.949,A -85,B 0,C 180,E1 -7295.958,E2 -7295.958} C_VEL
LIN {X 0,Y 474.049,Z 314.876,A -85,B 0,C 180,E1 -7297.453,E2 -7297.453} C_VEL
LIN {X 0,Y 474.377,Z 308.237,A -85,B 0,C 180,E1 -7298.734,E2 -7298.734} C_VEL
LIN {X 0,Y 474.75,Z 299.994,A -85,B 0,C 180,E1 -7300.017,E2 -7300.017} C_VEL
LIN {X 0,Y 475.092,Z 291.542,A -85,B 0,C 180,E1 -7301.087,E2 -7301.087} C_VEL
LIN {X 0,Y 475.625,Z 281.115,A -85,B 0,C 180,E1 -7302.153,E2 -7302.153} C_VEL
LIN {X 0,Y 476.024,Z 270.043,A -85,B 0,C 180,E1 -7303.065,E2 -7303.065} C_VEL
LIN {X 0,Y 476.438,Z 259.408,A -85,B 0,C 180,E1 -7303.76,E2 -7303.76} C_VEL
LIN {X 0,Y 476.931,Z 247.77,A -85,B 0,C 180,E1 -7304.344,E2 -7304.344} C_VEL
LIN {X 0,Y 476.842,Z 240.595,A -85,B 0,C 180,E1 -7304.633,E2 -7304.633} C_VEL
LIN {X 0,Y 474.723,Z 227.923,A -85,B 0,C 180,E1 -7305.073,E2 -7305.073} C_VEL
LIN {X 0,Y 474.117,Z 224.449,A -85,B 0,C 180,E1 -7305.172,E2 -7305.172} C_VEL
LIN {X 0,Y 474.282,Z 215.948,A -85,B 0,C 180,E1 -7308.492,E2 -7308.492} C_VEL
LIN {X 0,Y 474.454,Z 209.456,A -85,B 0,C 180,E1 -7311.059,E2 -7311.059} C_VEL
LIN {X 0,Y 474.669,Z 202.07,A -85,B 0,C 180,E1 -7314.027,E2 -7314.027} C_VEL
LIN {X 0,Y 474.94,Z 193.999,A -85,B 0,C 180,E1 -7317.394,E2 -7317.394} C_VEL
LIN {X 0,Y 475.202,Z 187.439,A -85,B 0,C 180,E1 -7320.188,E2 -7320.188} C_VEL
LIN {X 0,Y 475.432,Z 180.664,A -85,B 0,C 180,E1 -7323.157,E2 -7323.157} C_VEL
LIN {X 0,Y 475.599,Z 175.207,A -85,B 0,C 180,E1 -7325.635,E2 -7325.635} C_VEL
LIN {X 0,Y 475.039,Z 170.669,A -85,B 0,C 180,E1 -7327.829,E2 -7327.829} C_VEL
LIN {X 0,Y 474.633,Z 168.367,A -85,B 0,C 180,E1 -7328.999,E2 -7328.999} C_VEL
LIN {X 0,Y 474.624,Z 168.366,A -85,B 0,C 180,E1 -7332.236,E2 -7332.236} C_VEL
LIN {X 0,Y 474.616,Z 168.366,A -85,B 0,C 180,E1 -7335.297,E2 -7335.297} C_VEL
LIN {X 0,Y 474.619,Z 168.364,A -85,B 0,C 180,E1 -7338.214,E2 -7338.214} C_VEL
LIN {X 0,Y 474.628,Z 168.366,A -85,B 0,C 180,E1 -7340.452,E2 -7340.452} C_VEL
LIN {X 0,Y 474.572,Z 168.369,A -85,B 0,C 180,E1 -7343.675,E2 -7343.675} C_VEL
LIN {X 0,Y 474.632,Z 168.363,A -85,B 0,C 180,E1 -7346.779,E2 -7346.779} C_VEL
LIN {X 0,Y 474.604,Z 168.367,A -85,B 0,C 180,E1 -7349.77,E2 -7349.77} C_VEL
LIN {X 0,Y 474.695,Z 168.355,A -85,B 0,C 180,E1 -7352.68,E2 -7352.68} C_VEL
LIN {X 0,Y 474.638,Z 168.361,A -85,B 0,C 180,E1 -7355.506,E2 -7355.506} C_VEL
LIN {X 0,Y 474.668,Z 168.358,A -85,B 0,C 180,E1 -7359.185,E2 -7359.185} C_VEL
LIN {X 0,Y 474.653,Z 168.36,A -85,B 0,C 180,E1 -7361.884,E2 -7361.884} C_VEL
LIN {X 0,Y 474.698,Z 168.355,A -85,B 0,C 180,E1 -7364.544,E2 -7364.544} C_VEL
LIN {X 0,Y 474.702,Z 168.355,A -85,B 0,C 180,E1 -7368.038,E2 -7368.038} C_VEL
LIN {X 0,Y 474.693,Z 168.357,A -85,B 0,C 180,E1 -7371.486,E2 -7371.486} C_VEL
LIN {X 0,Y 474.745,Z 168.346,A -85,B 0,C 180,E1 -7374.052,E2 -7374.052} C_VEL
LIN {X 0,Y 474.89,Z 168.33,A -85,B 0,C 180,E1 -7377.455,E2 -7377.455} C_VEL
LIN {X 0,Y 474.91,Z 168.329,A -85,B 0,C 180,E1 -7380,E2 -7380} C_VEL
LIN {X 0,Y 474.89,Z 168.331,A -85,B 0,C 180,E1 -7382.545,E2 -7382.545} C_VEL
LIN {X 0,Y 474.744,Z 168.348,A -85,B 0,C 180,E1 -7385.948,E2 -7385.948} C_VEL
LIN {X 0,Y 474.693,Z 168.359,A -85,B 0,C 180,E1 -7388.514,E2 -7388.514} C_VEL
LIN {X 0,Y 474.702,Z 168.356,A -85,B 0,C 180,E1 -7391.963,E2 -7391.963} C_VEL
LIN {X 0,Y 474.698,Z 168.355,A -85,B 0,C 180,E1 -7395.456,E2 -7395.456} C_VEL
LIN {X 0,Y 474.663,Z 168.359,A -85,B 0,C 180,E1 -7399.01,E2 -7399.01} C_VEL
LIN {X 0,Y 474.586,Z 168.369,A -85,B 0,C 180,E1 -7401.729,E2 -7401.729} C_VEL
LIN {X 0,Y 474.639,Z 168.36,A -85,B 0,C 180,E1 -7404.494,E2 -7404.494} C_VEL
LIN {X 0,Y 474.698,Z 168.356,A -85,B 0,C 180,E1 -7407.339,E2 -7407.339} C_VEL
LIN {X 0,Y 474.603,Z 168.367,A -85,B 0,C 180,E1 -7410.81,E2 -7410.81} C_VEL
LIN {X 0,Y 474.635,Z 168.364,A -85,B 0,C 180,E1 -7413.984,E2 -7413.984} C_VEL
LIN {X 0,Y 474.551,Z 168.372,A -85,B 0,C 180,E1 -7416.897,E2 -7416.897} C_VEL
LIN {X 0,Y 474.613,Z 168.365,A -85,B 0,C 180,E1 -7419.646,E2 -7419.646} C_VEL
LIN {X 0,Y 474.623,Z 168.362,A -85,B 0,C 180,E1 -7422.237,E2 -7422.237} C_VEL
LIN {X 0,Y 474.621,Z 168.364,A -85,B 0,C 180,E1 -7425.298,E2 -7425.298} C_VEL
LIN {X 0,Y 474.62,Z 168.366,A -85,B 0,C 180,E1 -7428.215,E2 -7428.215} C_VEL
LIN {X 0,Y 474.607,Z 168.366,A -85,B 0,C 180,E1 -7431.543,E2 -7431.543} C_VEL
LIN {X 0,Y 474.462,Z 168.445,A -85,B 0,C 180,E1 -7434.557,E2 -7434.557} C_VEL
LIN {X 0,Y 474.448,Z 171.486,A -85,B 0,C 180,E1 -7436.765,E2 -7436.765} C_VEL
LIN {X 0,Y 474.383,Z 175.692,A -85,B 0,C 180,E1 -7439.755,E2 -7439.755} C_VEL
LIN {X 0,Y 474.277,Z 180.037,A -85,B 0,C 180,E1 -7442.761,E2 -7442.761} C_VEL
LIN {X 0,Y 474.199,Z 184.039,A -85,B 0,C 180,E1 -7445.482,E2 -7445.482} C_VEL
LIN {X 0,Y 474.098,Z 188.181,A -85,B 0,C 180,E1 -7448.248,E2 -7448.248} C_VEL
LIN {X 0,Y 473.972,Z 192.975,A -85,B 0,C 180,E1 -7451.334,E2 -7451.334} C_VEL
LIN {X 0,Y 473.28,Z 193.77,A -85,B 0,C 180,E1 -7451.797,E2 -7451.797} C_VEL
LIN {X 0,Y 470.389,Z 195.169,A -85,B 0,C 180,E1 -7452.515,E2 -7452.515} C_VEL
LIN {X 0,Y 467.493,Z 196.582,A -85,B 0,C 180,E1 -7453.242,E2 -7453.242} C_VEL
LIN {X 0,Y 466.814,Z 197.398,A -85,B 0,C 180,E1 -7453.714,E2 -7453.714} C_VEL
LIN {X 0,Y 466.87,Z 199.095,A -85,B 0,C 180,E1 -7454.676,E2 -7454.676} C_VEL
LIN {X 0,Y 469.686,Z 212.561,A -85,B 0,C 180,E1 -7455.163,E2 -7455.163} C_VEL
LIN {X 0,Y 470.256,Z 216.637,A -85,B 0,C 180,E1 -7455.337,E2 -7455.337} C_VEL
LIN {X 0,Y 469.846,Z 229.186,A -85,B 0,C 180,E1 -7455.933,E2 -7455.933} C_VEL
LIN {X 0,Y 469.329,Z 241.234,A -85,B 0,C 180,E1 -7456.692,E2 -7456.692} C_VEL
LIN {X 0,Y 468.943,Z 251.89,A -85,B 0,C 180,E1 -7457.559,E2 -7457.559} C_VEL
LIN {X 0,Y 468.468,Z 261.615,A -85,B 0,C 180,E1 -7458.535,E2 -7458.535} C_VEL
LIN {X 0,Y 468.014,Z 270.461,A -85,B 0,C 180,E1 -7459.619,E2 -7459.619} C_VEL
LIN {X 0,Y 467.578,Z 279.091,A -85,B 0,C 180,E1 -7460.92,E2 -7460.92} C_VEL
LIN {X 0,Y 467.22,Z 285.969,A -85,B 0,C 180,E1 -7462.22,E2 -7462.22} C_VEL
LIN {X 0,Y 467.04,Z 291.702,A -85,B 0,C 180,E1 -7463.582,E2 -7463.582} C_VEL
LIN {X 0,Y 466.803,Z 295.799,A -85,B 0,C 180,E1 -7464.817,E2 -7464.817} C_VEL
LIN {X 0,Y 466.784,Z 298.084,A -85,B 0,C 180,E1 -7465.683,E2 -7465.683} C_VEL
LIN {X 0,Y 466.796,Z 299.944,A -85,B 0,C 180,E1 -7466.548,E2 -7466.548} C_VEL
LIN {X 0,Y 466.693,Z 301.349,A -85,B 0,C 180,E1 -7467.411,E2 -7467.411} C_VEL
LIN {X 0,Y 466.621,Z 302.962,A -85,B 0,C 180,E1 -7469.137,E2 -7469.137} C_VEL
LIN {X 0,Y 466.601,Z 303.198,A -85,B 0,C 180,E1 -7470,E2 -7470} C_VEL
LIN {X 0,Y 466.621,Z 303.012,A -85,B 0,C 180,E1 -7470.863,E2 -7470.863} C_VEL
LIN {X 0,Y 466.693,Z 301.463,A -85,B 0,C 180,E1 -7472.59,E2 -7472.59} C_VEL
LIN {X 0,Y 466.796,Z 300.107,A -85,B 0,C 180,E1 -7473.453,E2 -7473.453} C_VEL
LIN {X 0,Y 466.752,Z 297.249,A -85,B 0,C 180,E1 -7474.751,E2 -7474.751} C_VEL
LIN {X 0,Y 467.015,Z 293.363,A -85,B 0,C 180,E1 -7476.047,E2 -7476.047} C_VEL
LIN {X 0,Y 467.103,Z 288.358,A -85,B 0,C 180,E1 -7477.348,E2 -7477.348} C_VEL
LIN {X 0,Y 467.425,Z 282.052,A -85,B 0,C 180,E1 -7478.648,E2 -7478.648} C_VEL
LIN {X 0,Y 467.813,Z 274.157,A -85,B 0,C 180,E1 -7479.949,E2 -7479.949} C_VEL
LIN {X 0,Y 468.206,Z 266.109,A -85,B 0,C 180,E1 -7481.034,E2 -7481.034} C_VEL
LIN {X 0,Y 468.727,Z 256.285,A -85,B 0,C 180,E1 -7482.117,E2 -7482.117} C_VEL
LIN {X 0,Y 469.171,Z 245.246,A -85,B 0,C 180,E1 -7483.095,E2 -7483.095} C_VEL
LIN {X 0,Y 469.652,Z 234.411,A -85,B 0,C 180,E1 -7483.853,E2 -7483.853} C_VEL
LIN {X 0,Y 470.095,Z 222.449,A -85,B 0,C 180,E1 -7484.502,E2 -7484.502} C_VEL
LIN {X 0,Y 470.167,Z 215.36,A -85,B 0,C 180,E1 -7484.811,E2 -7484.811} C_VEL
LIN {X 0,Y 467.667,Z 202.838,A -85,B 0,C 180,E1 -7485.298,E2 -7485.298} C_VEL
LIN {X 0,Y 466.84,Z 198.911,A -85,B 0,C 180,E1 -7485.441,E2 -7485.441} C_VEL
LIN {X 0,Y 466.916,Z 194.013,A -85,B 0,C 180,E1 -7488.508,E2 -7488.508} C_VEL
LIN {X 0,Y 466.989,Z 189.903,A -85,B 0,C 180,E1 -7491.173,E2 -7491.173} C_VEL
LIN {X 0,Y 467.113,Z 185.724,A -85,B 0,C 180,E1 -7493.968,E2 -7493.968} C_VEL
LIN {X 0,Y 467.177,Z 181.561,A -85,B 0,C 180,E1 -7496.828,E2 -7496.828} C_VEL
LIN {X 0,Y 467.33,Z 177.361,A -85,B 0,C 180,E1 -7499.754,E2 -7499.754} C_VEL
LIN {X 0,Y 467.395,Z 173.127,A -85,B 0,C 180,E1 -7502.773,E2 -7502.773} C_VEL
LIN {X 0,Y 467.468,Z 170.305,A -85,B 0,C 180,E1 -7504.841,E2 -7504.841} C_VEL
LIN {X 0,Y 467.482,Z 169.256,A -85,B 0,C 180,E1 -7505.896,E2 -7505.896} C_VEL
LIN {X 0,Y 467.543,Z 169.248,A -85,B 0,C 180,E1 -7509.149,E2 -7509.149} C_VEL
LIN {X 0,Y 467.566,Z 169.243,A -85,B 0,C 180,E1 -7511.404,E2 -7511.404} C_VEL
LIN {X 0,Y 467.567,Z 169.244,A -85,B 0,C 180,E1 -7515.052,E2 -7515.052} C_VEL
LIN {X 0,Y 467.591,Z 169.24,A -85,B 0,C 180,E1 -7517.44,E2 -7517.44} C_VEL
LIN {X 0,Y 467.552,Z 169.247,A -85,B 0,C 180,E1 -7520.852,E2 -7520.852} C_VEL
LIN {X 0,Y 467.552,Z 169.247,A -85,B 0,C 180,E1 -7524.262,E2 -7524.262} C_VEL
LIN {X 0,Y 467.58,Z 169.242,A -85,B 0,C 180,E1 -7527.321,E2 -7527.321} C_VEL
LIN {X 0,Y 467.572,Z 169.245,A -85,B 0,C 180,E1 -7530.667,E2 -7530.667} C_VEL
LIN {X 0,Y 467.614,Z 169.235,A -85,B 0,C 180,E1 -7533.199,E2 -7533.199} C_VEL
LIN {X 0,Y 467.592,Z 169.24,A -85,B 0,C 180,E1 -7536.469,E2 -7536.469} C_VEL
LIN {X 0,Y 467.623,Z 169.239,A -85,B 0,C 180,E1 -7539.777,E2 -7539.777} C_VEL
LIN {X 0,Y 467.6,Z 169.24,A -85,B 0,C 180,E1 -7542.506,E2 -7542.506} C_VEL
LIN {X 0,Y 467.607,Z 169.239,A -85,B 0,C 180,E1 -7545.196,E2 -7545.196} C_VEL
LIN {X 0,Y 467.657,Z 169.234,A -85,B 0,C 180,E1 -7547.854,E2 -7547.854} C_VEL
LIN {X 0,Y 467.657,Z 169.233,A -85,B 0,C 180,E1 -7551.357,E2 -7551.357} C_VEL
LIN {X 0,Y 467.709,Z 169.224,A -85,B 0,C 180,E1 -7553.962,E2 -7553.962} C_VEL
LIN {X 0,Y 467.857,Z 169.207,A -85,B 0,C 180,E1 -7557.417,E2 -7557.417} C_VEL
LIN {X 0,Y 467.884,Z 169.204,A -85,B 0,C 180,E1 -7560,E2 -7560} C_VEL
LIN {X 0,Y 467.858,Z 169.206,A -85,B 0,C 180,E1 -7562.583,E2 -7562.583} C_VEL
LIN {X 0,Y 467.711,Z 169.222,A -85,B 0,C 180,E1 -7566.038,E2 -7566.038} C_VEL
LIN {X 0,Y 467.656,Z 169.235,A -85,B 0,C 180,E1 -7568.643,E2 -7568.643} C_VEL
LIN {X 0,Y 467.683,Z 169.23,A -85,B 0,C 180,E1 -7572.145,E2 -7572.145} C_VEL
LIN {X 0,Y 467.65,Z 169.234,A -85,B 0,C 180,E1 -7575.885,E2 -7575.885} C_VEL
LIN {X 0,Y 467.623,Z 169.235,A -85,B 0,C 180,E1 -7579.308,E2 -7579.308} C_VEL
LIN {X 0,Y 467.535,Z 169.248,A -85,B 0,C 180,E1 -7582.074,E2 -7582.074} C_VEL
LIN {X 0,Y 467.585,Z 169.239,A -85,B 0,C 180,E1 -7584.888,E2 -7584.888} C_VEL
LIN {X 0,Y 467.621,Z 169.239,A -85,B 0,C 180,E1 -7587.769,E2 -7587.769} C_VEL
LIN {X 0,Y 467.569,Z 169.243,A -85,B 0,C 180,E1 -7591.045,E2 -7591.045} C_VEL
LIN {X 0,Y 467.588,Z 169.241,A -85,B 0,C 180,E1 -7594.242,E2 -7594.242} C_VEL
LIN {X 0,Y 467.516,Z 169.248,A -85,B 0,C 180,E1 -7597.181,E2 -7597.181} C_VEL
LIN {X 0,Y 467.574,Z 169.24,A -85,B 0,C 180,E1 -7600.265,E2 -7600.265} C_VEL
LIN {X 0,Y 467.588,Z 169.24,A -85,B 0,C 180,E1 -7602.567,E2 -7602.567} C_VEL
LIN {X 0,Y 467.567,Z 169.244,A -85,B 0,C 180,E1 -7605.053,E2 -7605.053} C_VEL
LIN {X 0,Y 467.59,Z 169.239,A -85,B 0,C 180,E1 -7607.44,E2 -7607.44} C_VEL
LIN {X 0,Y 467.611,Z 169.39,A -85,B 0,C 180,E1 -7610.858,E2 -7610.858} C_VEL
LIN {X 0,Y 468.483,Z 174.95,A -85,B 0,C 180,E1 -7613.651,E2 -7613.651} C_VEL
LIN {X 0,Y 468.562,Z 179.037,A -85,B 0,C 180,E1 -7615.584,E2 -7615.584} C_VEL
LIN {X 0,Y 468.245,Z 186.209,A -85,B 0,C 180,E1 -7618.818,E2 -7618.818} C_VEL
LIN {X 0,Y 468,Z 192.967,A -85,B 0,C 180,E1 -7621.768,E2 -7621.768} C_VEL
LIN {X 0,Y 467.671,Z 200.848,A -85,B 0,C 180,E1 -7625.116,E2 -7625.116} C_VEL
LIN {X 0,Y 467.464,Z 207.664,A -85,B 0,C 180,E1 -7627.923,E2 -7627.923} C_VEL
LIN {X 0,Y 467.308,Z 214.483,A -85,B 0,C 180,E1 -7630.679,E2 -7630.679} C_VEL
LIN {X 0,Y 467.099,Z 223.717,A -85,B 0,C 180,E1 -7634.355,E2 -7634.355} C_VEL
LIN {X 0,Y 467.076,Z 224.336,A -85,B 0,C 180,E1 -7634.599,E2 -7634.599} C_VEL
LIN {X 0,Y 469.5,Z 238.076,A -85,B 0,C 180,E1 -7635.048,E2 -7635.048} C_VEL
LIN {X 0,Y 470.158,Z 243.714,A -85,B 0,C 180,E1 -7635.278,E2 -7635.278} C_VEL
LIN {X 0,Y 469.76,Z 255.367,A -85,B 0,C 180,E1 -7635.819,E2 -7635.819} C_VEL
LIN {X 0,Y 469.269,Z 266.568,A -85,B 0,C 180,E1 -7636.5,E2 -7636.5} C_VEL
LIN {X 0,Y 468.806,Z 277.389,A -85,B 0,C 180,E1 -7637.333,E2 -7637.333} C_VEL
LIN {X 0,Y 468.389,Z 287.612,A -85,B 0,C 180,E1 -7638.313,E2 -7638.313} C_VEL
